FUNCTION_BLOCK "UNI_TO_GB2"   // FB9, SCL
{ S7_Optimized_Access := 'TRUE' }
VERSION : 0.1
   VAR_INPUT
      UNICODE : Word;
   END_VAR
   VAR_OUTPUT
      GB2312 : Word;
   END_VAR
   VAR
      UNI : Array[0..7480] of Word;
      GB2 : Array[0..7480] of Word;
   END_VAR
   VAR_TEMP
      i : UDInt;
      j : UDInt;
      li : UDInt;
      hi : UDInt;
   END_VAR
   // UNI[0] := 16#00A4;
   // UNI[1] := 16#00A7;
   // UNI[2] := 16#00A8;
   // UNI[3] := 16#00B0;
   // UNI[4] := 16#00B1;
   // UNI[5] := 16#00B7;
   // UNI[6] := 16#00D7;
   // UNI[7] := 16#00E0;
   // UNI[8] := 16#00E1;
   // UNI[9] := 16#00E8;
   // UNI[10] := 16#00E9;
   // UNI[11] := 16#00EA;
   // UNI[12] := 16#00EC;
   // UNI[13] := 16#00ED;
   // UNI[14] := 16#00F2;
   // UNI[15] := 16#00F3;
   // UNI[16] := 16#00F7;
   // UNI[17] := 16#00F9;
   // UNI[18] := 16#00FA;
   // UNI[19] := 16#00FC;
   // UNI[20] := 16#0101;
   // UNI[21] := 16#0113;
   // UNI[22] := 16#011B;
   // UNI[23] := 16#012B;
   // UNI[24] := 16#0144;
   // UNI[25] := 16#0148;
   // UNI[26] := 16#014D;
   // UNI[27] := 16#016B;
   // UNI[28] := 16#01CE;
   // UNI[29] := 16#01D0;
   // UNI[30] := 16#01D2;
   // UNI[31] := 16#01D4;
   // UNI[32] := 16#01D6;
   // UNI[33] := 16#01D8;
   // UNI[34] := 16#01DA;
   // UNI[35] := 16#01DC;
   // UNI[36] := 16#0251;
   // UNI[37] := 16#0261;
   // UNI[38] := 16#02C7;
   // UNI[39] := 16#02C9;
   // UNI[40] := 16#0391;
   // UNI[41] := 16#0392;
   // UNI[42] := 16#0393;
   // UNI[43] := 16#0394;
   // UNI[44] := 16#0395;
   // UNI[45] := 16#0396;
   // UNI[46] := 16#0397;
   // UNI[47] := 16#0398;
   // UNI[48] := 16#0399;
   // UNI[49] := 16#039A;
   // UNI[50] := 16#039B;
   // UNI[51] := 16#039C;
   // UNI[52] := 16#039D;
   // UNI[53] := 16#039E;
   // UNI[54] := 16#039F;
   // UNI[55] := 16#03A0;
   // UNI[56] := 16#03A1;
   // UNI[57] := 16#03A3;
   // UNI[58] := 16#03A4;
   // UNI[59] := 16#03A5;
   // UNI[60] := 16#03A6;
   // UNI[61] := 16#03A7;
   // UNI[62] := 16#03A8;
   // UNI[63] := 16#03A9;
   // UNI[64] := 16#03B1;
   // UNI[65] := 16#03B2;
   // UNI[66] := 16#03B3;
   // UNI[67] := 16#03B4;
   // UNI[68] := 16#03B5;
   // UNI[69] := 16#03B6;
   // UNI[70] := 16#03B7;
   // UNI[71] := 16#03B8;
   // UNI[72] := 16#03B9;
   // UNI[73] := 16#03BA;
   // UNI[74] := 16#03BB;
   // UNI[75] := 16#03BC;
   // UNI[76] := 16#03BD;
   // UNI[77] := 16#03BE;
   // UNI[78] := 16#03BF;
   // UNI[79] := 16#03C0;
   // UNI[80] := 16#03C1;
   // UNI[81] := 16#03C3;
   // UNI[82] := 16#03C4;
   // UNI[83] := 16#03C5;
   // UNI[84] := 16#03C6;
   // UNI[85] := 16#03C7;
   // UNI[86] := 16#03C8;
   // UNI[87] := 16#03C9;
   // UNI[88] := 16#0401;
   // UNI[89] := 16#0410;
   // UNI[90] := 16#0411;
   // UNI[91] := 16#0412;
   // UNI[92] := 16#0413;
   // UNI[93] := 16#0414;
   // UNI[94] := 16#0415;
   // UNI[95] := 16#0416;
   // UNI[96] := 16#0417;
   // UNI[97] := 16#0418;
   // UNI[98] := 16#0419;
   // UNI[99] := 16#041A;
   // UNI[100] := 16#041B;
   // UNI[101] := 16#041C;
   // UNI[102] := 16#041D;
   // UNI[103] := 16#041E;
   // UNI[104] := 16#041F;
   // UNI[105] := 16#0420;
   // UNI[106] := 16#0421;
   // UNI[107] := 16#0422;
   // UNI[108] := 16#0423;
   // UNI[109] := 16#0424;
   // UNI[110] := 16#0425;
   // UNI[111] := 16#0426;
   // UNI[112] := 16#0427;
   // UNI[113] := 16#0428;
   // UNI[114] := 16#0429;
   // UNI[115] := 16#042A;
   // UNI[116] := 16#042B;
   // UNI[117] := 16#042C;
   // UNI[118] := 16#042D;
   // UNI[119] := 16#042E;
   // UNI[120] := 16#042F;
   // UNI[121] := 16#0430;
   // UNI[122] := 16#0431;
   // UNI[123] := 16#0432;
   // UNI[124] := 16#0433;
   // UNI[125] := 16#0434;
   // UNI[126] := 16#0435;
   // UNI[127] := 16#0436;
   // UNI[128] := 16#0437;
   // UNI[129] := 16#0438;
   // UNI[130] := 16#0439;
   // UNI[131] := 16#043A;
   // UNI[132] := 16#043B;
   // UNI[133] := 16#043C;
   // UNI[134] := 16#043D;
   // UNI[135] := 16#043E;
   // UNI[136] := 16#043F;
   // UNI[137] := 16#0440;
   // UNI[138] := 16#0441;
   // UNI[139] := 16#0442;
   // UNI[140] := 16#0443;
   // UNI[141] := 16#0444;
   // UNI[142] := 16#0445;
   // UNI[143] := 16#0446;
   // UNI[144] := 16#0447;
   // UNI[145] := 16#0448;
   // UNI[146] := 16#0449;
   // UNI[147] := 16#044A;
   // UNI[148] := 16#044B;
   // UNI[149] := 16#044C;
   // UNI[150] := 16#044D;
   // UNI[151] := 16#044E;
   // UNI[152] := 16#044F;
   // UNI[153] := 16#0451;
   // UNI[154] := 16#2014;
   // UNI[155] := 16#2016;
   // UNI[156] := 16#2018;
   // UNI[157] := 16#2019;
   // UNI[158] := 16#201C;
   // UNI[159] := 16#201D;
   // UNI[160] := 16#2026;
   // UNI[161] := 16#2030;
   // UNI[162] := 16#2032;
   // UNI[163] := 16#2033;
   // UNI[164] := 16#203B;
   // UNI[165] := 16#2103;
   // UNI[166] := 16#2116;
   // UNI[167] := 16#2160;
   // UNI[168] := 16#2161;
   // UNI[169] := 16#2162;
   // UNI[170] := 16#2163;
   // UNI[171] := 16#2164;
   // UNI[172] := 16#2165;
   // UNI[173] := 16#2166;
   // UNI[174] := 16#2167;
   // UNI[175] := 16#2168;
   // UNI[176] := 16#2169;
   // UNI[177] := 16#216A;
   // UNI[178] := 16#216B;
   // UNI[179] := 16#2170;
   // UNI[180] := 16#2171;
   // UNI[181] := 16#2172;
   // UNI[182] := 16#2173;
   // UNI[183] := 16#2174;
   // UNI[184] := 16#2175;
   // UNI[185] := 16#2176;
   // UNI[186] := 16#2177;
   // UNI[187] := 16#2178;
   // UNI[188] := 16#2179;
   // UNI[189] := 16#2190;
   // UNI[190] := 16#2191;
   // UNI[191] := 16#2192;
   // UNI[192] := 16#2193;
   // UNI[193] := 16#2208;
   // UNI[194] := 16#220F;
   // UNI[195] := 16#2211;
   // UNI[196] := 16#221A;
   // UNI[197] := 16#221D;
   // UNI[198] := 16#221E;
   // UNI[199] := 16#2220;
   // UNI[200] := 16#2225;
   // UNI[201] := 16#2227;
   // UNI[202] := 16#2228;
   // UNI[203] := 16#2229;
   // UNI[204] := 16#222A;
   // UNI[205] := 16#222B;
   // UNI[206] := 16#222E;
   // UNI[207] := 16#2234;
   // UNI[208] := 16#2235;
   // UNI[209] := 16#2236;
   // UNI[210] := 16#2237;
   // UNI[211] := 16#223D;
   // UNI[212] := 16#2248;
   // UNI[213] := 16#224C;
   // UNI[214] := 16#2260;
   // UNI[215] := 16#2261;
   // UNI[216] := 16#2264;
   // UNI[217] := 16#2265;
   // UNI[218] := 16#226E;
   // UNI[219] := 16#226F;
   // UNI[220] := 16#2299;
   // UNI[221] := 16#22A5;
   // UNI[222] := 16#2312;
   // UNI[223] := 16#2460;
   // UNI[224] := 16#2461;
   // UNI[225] := 16#2462;
   // UNI[226] := 16#2463;
   // UNI[227] := 16#2464;
   // UNI[228] := 16#2465;
   // UNI[229] := 16#2466;
   // UNI[230] := 16#2467;
   // UNI[231] := 16#2468;
   // UNI[232] := 16#2469;
   // UNI[233] := 16#2474;
   // UNI[234] := 16#2475;
   // UNI[235] := 16#2476;
   // UNI[236] := 16#2477;
   // UNI[237] := 16#2478;
   // UNI[238] := 16#2479;
   // UNI[239] := 16#247A;
   // UNI[240] := 16#247B;
   // UNI[241] := 16#247C;
   // UNI[242] := 16#247D;
   // UNI[243] := 16#247E;
   // UNI[244] := 16#247F;
   // UNI[245] := 16#2480;
   // UNI[246] := 16#2481;
   // UNI[247] := 16#2482;
   // UNI[248] := 16#2483;
   // UNI[249] := 16#2484;
   // UNI[250] := 16#2485;
   // UNI[251] := 16#2486;
   // UNI[252] := 16#2487;
   // UNI[253] := 16#2488;
   // UNI[254] := 16#2489;
   // UNI[255] := 16#248A;
   // UNI[256] := 16#248B;
   // UNI[257] := 16#248C;
   // UNI[258] := 16#248D;
   // UNI[259] := 16#248E;
   // UNI[260] := 16#248F;
   // UNI[261] := 16#2490;
   // UNI[262] := 16#2491;
   // UNI[263] := 16#2492;
   // UNI[264] := 16#2493;
   // UNI[265] := 16#2494;
   // UNI[266] := 16#2495;
   // UNI[267] := 16#2496;
   // UNI[268] := 16#2497;
   // UNI[269] := 16#2498;
   // UNI[270] := 16#2499;
   // UNI[271] := 16#249A;
   // UNI[272] := 16#249B;
   // UNI[273] := 16#2500;
   // UNI[274] := 16#2501;
   // UNI[275] := 16#2502;
   // UNI[276] := 16#2503;
   // UNI[277] := 16#2504;
   // UNI[278] := 16#2505;
   // UNI[279] := 16#2506;
   // UNI[280] := 16#2507;
   // UNI[281] := 16#2508;
   // UNI[282] := 16#2509;
   // UNI[283] := 16#250A;
   // UNI[284] := 16#250B;
   // UNI[285] := 16#250C;
   // UNI[286] := 16#250D;
   // UNI[287] := 16#250E;
   // UNI[288] := 16#250F;
   // UNI[289] := 16#2510;
   // UNI[290] := 16#2511;
   // UNI[291] := 16#2512;
   // UNI[292] := 16#2513;
   // UNI[293] := 16#2514;
   // UNI[294] := 16#2515;
   // UNI[295] := 16#2516;
   // UNI[296] := 16#2517;
   // UNI[297] := 16#2518;
   // UNI[298] := 16#2519;
   // UNI[299] := 16#251A;
   // UNI[300] := 16#251B;
   // UNI[301] := 16#251C;
   // UNI[302] := 16#251D;
   // UNI[303] := 16#251E;
   // UNI[304] := 16#251F;
   // UNI[305] := 16#2520;
   // UNI[306] := 16#2521;
   // UNI[307] := 16#2522;
   // UNI[308] := 16#2523;
   // UNI[309] := 16#2524;
   // UNI[310] := 16#2525;
   // UNI[311] := 16#2526;
   // UNI[312] := 16#2527;
   // UNI[313] := 16#2528;
   // UNI[314] := 16#2529;
   // UNI[315] := 16#252A;
   // UNI[316] := 16#252B;
   // UNI[317] := 16#252C;
   // UNI[318] := 16#252D;
   // UNI[319] := 16#252E;
   // UNI[320] := 16#252F;
   // UNI[321] := 16#2530;
   // UNI[322] := 16#2531;
   // UNI[323] := 16#2532;
   // UNI[324] := 16#2533;
   // UNI[325] := 16#2534;
   // UNI[326] := 16#2535;
   // UNI[327] := 16#2536;
   // UNI[328] := 16#2537;
   // UNI[329] := 16#2538;
   // UNI[330] := 16#2539;
   // UNI[331] := 16#253A;
   // UNI[332] := 16#253B;
   // UNI[333] := 16#253C;
   // UNI[334] := 16#253D;
   // UNI[335] := 16#253E;
   // UNI[336] := 16#253F;
   // UNI[337] := 16#2540;
   // UNI[338] := 16#2541;
   // UNI[339] := 16#2542;
   // UNI[340] := 16#2543;
   // UNI[341] := 16#2544;
   // UNI[342] := 16#2545;
   // UNI[343] := 16#2546;
   // UNI[344] := 16#2547;
   // UNI[345] := 16#2548;
   // UNI[346] := 16#2549;
   // UNI[347] := 16#254A;
   // UNI[348] := 16#254B;
   // UNI[349] := 16#25A0;
   // UNI[350] := 16#25A1;
   // UNI[351] := 16#25B2;
   // UNI[352] := 16#25B3;
   // UNI[353] := 16#25C6;
   // UNI[354] := 16#25C7;
   // UNI[355] := 16#25CB;
   // UNI[356] := 16#25CE;
   // UNI[357] := 16#25CF;
   // UNI[358] := 16#2605;
   // UNI[359] := 16#2606;
   // UNI[360] := 16#2640;
   // UNI[361] := 16#2642;
   // UNI[362] := 16#3000;
   // UNI[363] := 16#3001;
   // UNI[364] := 16#3002;
   // UNI[365] := 16#3003;
   // UNI[366] := 16#3005;
   // UNI[367] := 16#3008;
   // UNI[368] := 16#3009;
   // UNI[369] := 16#300A;
   // UNI[370] := 16#300B;
   // UNI[371] := 16#300C;
   // UNI[372] := 16#300D;
   // UNI[373] := 16#300E;
   // UNI[374] := 16#300F;
   // UNI[375] := 16#3010;
   // UNI[376] := 16#3011;
   // UNI[377] := 16#3013;
   // UNI[378] := 16#3014;
   // UNI[379] := 16#3015;
   // UNI[380] := 16#3016;
   // UNI[381] := 16#3017;
   // UNI[382] := 16#3041;
   // UNI[383] := 16#3042;
   // UNI[384] := 16#3043;
   // UNI[385] := 16#3044;
   // UNI[386] := 16#3045;
   // UNI[387] := 16#3046;
   // UNI[388] := 16#3047;
   // UNI[389] := 16#3048;
   // UNI[390] := 16#3049;
   // UNI[391] := 16#304A;
   // UNI[392] := 16#304B;
   // UNI[393] := 16#304C;
   // UNI[394] := 16#304D;
   // UNI[395] := 16#304E;
   // UNI[396] := 16#304F;
   // UNI[397] := 16#3050;
   // UNI[398] := 16#3051;
   // UNI[399] := 16#3052;
   // UNI[400] := 16#3053;
   // UNI[401] := 16#3054;
   // UNI[402] := 16#3055;
   // UNI[403] := 16#3056;
   // UNI[404] := 16#3057;
   // UNI[405] := 16#3058;
   // UNI[406] := 16#3059;
   // UNI[407] := 16#305A;
   // UNI[408] := 16#305B;
   // UNI[409] := 16#305C;
   // UNI[410] := 16#305D;
   // UNI[411] := 16#305E;
   // UNI[412] := 16#305F;
   // UNI[413] := 16#3060;
   // UNI[414] := 16#3061;
   // UNI[415] := 16#3062;
   // UNI[416] := 16#3063;
   // UNI[417] := 16#3064;
   // UNI[418] := 16#3065;
   // UNI[419] := 16#3066;
   // UNI[420] := 16#3067;
   // UNI[421] := 16#3068;
   // UNI[422] := 16#3069;
   // UNI[423] := 16#306A;
   // UNI[424] := 16#306B;
   // UNI[425] := 16#306C;
   // UNI[426] := 16#306D;
   // UNI[427] := 16#306E;
   // UNI[428] := 16#306F;
   // UNI[429] := 16#3070;
   // UNI[430] := 16#3071;
   // UNI[431] := 16#3072;
   // UNI[432] := 16#3073;
   // UNI[433] := 16#3074;
   // UNI[434] := 16#3075;
   // UNI[435] := 16#3076;
   // UNI[436] := 16#3077;
   // UNI[437] := 16#3078;
   // UNI[438] := 16#3079;
   // UNI[439] := 16#307A;
   // UNI[440] := 16#307B;
   // UNI[441] := 16#307C;
   // UNI[442] := 16#307D;
   // UNI[443] := 16#307E;
   // UNI[444] := 16#307F;
   // UNI[445] := 16#3080;
   // UNI[446] := 16#3081;
   // UNI[447] := 16#3082;
   // UNI[448] := 16#3083;
   // UNI[449] := 16#3084;
   // UNI[450] := 16#3085;
   // UNI[451] := 16#3086;
   // UNI[452] := 16#3087;
   // UNI[453] := 16#3088;
   // UNI[454] := 16#3089;
   // UNI[455] := 16#308A;
   // UNI[456] := 16#308B;
   // UNI[457] := 16#308C;
   // UNI[458] := 16#308D;
   // UNI[459] := 16#308E;
   // UNI[460] := 16#308F;
   // UNI[461] := 16#3090;
   // UNI[462] := 16#3091;
   // UNI[463] := 16#3092;
   // UNI[464] := 16#3093;
   // UNI[465] := 16#30A1;
   // UNI[466] := 16#30A2;
   // UNI[467] := 16#30A3;
   // UNI[468] := 16#30A4;
   // UNI[469] := 16#30A5;
   // UNI[470] := 16#30A6;
   // UNI[471] := 16#30A7;
   // UNI[472] := 16#30A8;
   // UNI[473] := 16#30A9;
   // UNI[474] := 16#30AA;
   // UNI[475] := 16#30AB;
   // UNI[476] := 16#30AC;
   // UNI[477] := 16#30AD;
   // UNI[478] := 16#30AE;
   // UNI[479] := 16#30AF;
   // UNI[480] := 16#30B0;
   // UNI[481] := 16#30B1;
   // UNI[482] := 16#30B2;
   // UNI[483] := 16#30B3;
   // UNI[484] := 16#30B4;
   // UNI[485] := 16#30B5;
   // UNI[486] := 16#30B6;
   // UNI[487] := 16#30B7;
   // UNI[488] := 16#30B8;
   // UNI[489] := 16#30B9;
   // UNI[490] := 16#30BA;
   // UNI[491] := 16#30BB;
   // UNI[492] := 16#30BC;
   // UNI[493] := 16#30BD;
   // UNI[494] := 16#30BE;
   // UNI[495] := 16#30BF;
   // UNI[496] := 16#30C0;
   // UNI[497] := 16#30C1;
   // UNI[498] := 16#30C2;
   // UNI[499] := 16#30C3;
   // UNI[500] := 16#30C4;
   // UNI[501] := 16#30C5;
   // UNI[502] := 16#30C6;
   // UNI[503] := 16#30C7;
   // UNI[504] := 16#30C8;
   // UNI[505] := 16#30C9;
   // UNI[506] := 16#30CA;
   // UNI[507] := 16#30CB;
   // UNI[508] := 16#30CC;
   // UNI[509] := 16#30CD;
   // UNI[510] := 16#30CE;
   // UNI[511] := 16#30CF;
   // UNI[512] := 16#30D0;
   // UNI[513] := 16#30D1;
   // UNI[514] := 16#30D2;
   // UNI[515] := 16#30D3;
   // UNI[516] := 16#30D4;
   // UNI[517] := 16#30D5;
   // UNI[518] := 16#30D6;
   // UNI[519] := 16#30D7;
   // UNI[520] := 16#30D8;
   // UNI[521] := 16#30D9;
   // UNI[522] := 16#30DA;
   // UNI[523] := 16#30DB;
   // UNI[524] := 16#30DC;
   // UNI[525] := 16#30DD;
   // UNI[526] := 16#30DE;
   // UNI[527] := 16#30DF;
   // UNI[528] := 16#30E0;
   // UNI[529] := 16#30E1;
   // UNI[530] := 16#30E2;
   // UNI[531] := 16#30E3;
   // UNI[532] := 16#30E4;
   // UNI[533] := 16#30E5;
   // UNI[534] := 16#30E6;
   // UNI[535] := 16#30E7;
   // UNI[536] := 16#30E8;
   // UNI[537] := 16#30E9;
   // UNI[538] := 16#30EA;
   // UNI[539] := 16#30EB;
   // UNI[540] := 16#30EC;
   // UNI[541] := 16#30ED;
   // UNI[542] := 16#30EE;
   // UNI[543] := 16#30EF;
   // UNI[544] := 16#30F0;
   // UNI[545] := 16#30F1;
   // UNI[546] := 16#30F2;
   // UNI[547] := 16#30F3;
   // UNI[548] := 16#30F4;
   // UNI[549] := 16#30F5;
   // UNI[550] := 16#30F6;
   // UNI[551] := 16#3105;
   // UNI[552] := 16#3106;
   // UNI[553] := 16#3107;
   // UNI[554] := 16#3108;
   // UNI[555] := 16#3109;
   // UNI[556] := 16#310A;
   // UNI[557] := 16#310B;
   // UNI[558] := 16#310C;
   // UNI[559] := 16#310D;
   // UNI[560] := 16#310E;
   // UNI[561] := 16#310F;
   // UNI[562] := 16#3110;
   // UNI[563] := 16#3111;
   // UNI[564] := 16#3112;
   // UNI[565] := 16#3113;
   // UNI[566] := 16#3114;
   // UNI[567] := 16#3115;
   // UNI[568] := 16#3116;
   // UNI[569] := 16#3117;
   // UNI[570] := 16#3118;
   // UNI[571] := 16#3119;
   // UNI[572] := 16#311A;
   // UNI[573] := 16#311B;
   // UNI[574] := 16#311C;
   // UNI[575] := 16#311D;
   // UNI[576] := 16#311E;
   // UNI[577] := 16#311F;
   // UNI[578] := 16#3120;
   // UNI[579] := 16#3121;
   // UNI[580] := 16#3122;
   // UNI[581] := 16#3123;
   // UNI[582] := 16#3124;
   // UNI[583] := 16#3125;
   // UNI[584] := 16#3126;
   // UNI[585] := 16#3127;
   // UNI[586] := 16#3128;
   // UNI[587] := 16#3129;
   // UNI[588] := 16#3220;
   // UNI[589] := 16#3221;
   // UNI[590] := 16#3222;
   // UNI[591] := 16#3223;
   // UNI[592] := 16#3224;
   // UNI[593] := 16#3225;
   // UNI[594] := 16#3226;
   // UNI[595] := 16#3227;
   // UNI[596] := 16#3228;
   // UNI[597] := 16#3229;
   // UNI[598] := 16#4E00;
   // UNI[599] := 16#4E01;
   // UNI[600] := 16#4E03;
   // UNI[601] := 16#4E07;
   // UNI[602] := 16#4E08;
   // UNI[603] := 16#4E09;
   // UNI[604] := 16#4E0A;
   // UNI[605] := 16#4E0B;
   // UNI[606] := 16#4E0C;
   // UNI[607] := 16#4E0D;
   // UNI[608] := 16#4E0E;
   // UNI[609] := 16#4E10;
   // UNI[610] := 16#4E11;
   // UNI[611] := 16#4E13;
   // UNI[612] := 16#4E14;
   // UNI[613] := 16#4E15;
   // UNI[614] := 16#4E16;
   // UNI[615] := 16#4E18;
   // UNI[616] := 16#4E19;
   // UNI[617] := 16#4E1A;
   // UNI[618] := 16#4E1B;
   // UNI[619] := 16#4E1C;
   // UNI[620] := 16#4E1D;
   // UNI[621] := 16#4E1E;
   // UNI[622] := 16#4E22;
   // UNI[623] := 16#4E24;
   // UNI[624] := 16#4E25;
   // UNI[625] := 16#4E27;
   // UNI[626] := 16#4E28;
   // UNI[627] := 16#4E2A;
   // UNI[628] := 16#4E2B;
   // UNI[629] := 16#4E2C;
   // UNI[630] := 16#4E2D;
   // UNI[631] := 16#4E30;
   // UNI[632] := 16#4E32;
   // UNI[633] := 16#4E34;
   // UNI[634] := 16#4E36;
   // UNI[635] := 16#4E38;
   // UNI[636] := 16#4E39;
   // UNI[637] := 16#4E3A;
   // UNI[638] := 16#4E3B;
   // UNI[639] := 16#4E3D;
   // UNI[640] := 16#4E3E;
   // UNI[641] := 16#4E3F;
   // UNI[642] := 16#4E43;
   // UNI[643] := 16#4E45;
   // UNI[644] := 16#4E47;
   // UNI[645] := 16#4E48;
   // UNI[646] := 16#4E49;
   // UNI[647] := 16#4E4B;
   // UNI[648] := 16#4E4C;
   // UNI[649] := 16#4E4D;
   // UNI[650] := 16#4E4E;
   // UNI[651] := 16#4E4F;
   // UNI[652] := 16#4E50;
   // UNI[653] := 16#4E52;
   // UNI[654] := 16#4E53;
   // UNI[655] := 16#4E54;
   // UNI[656] := 16#4E56;
   // UNI[657] := 16#4E58;
   // UNI[658] := 16#4E59;
   // UNI[659] := 16#4E5C;
   // UNI[660] := 16#4E5D;
   // UNI[661] := 16#4E5E;
   // UNI[662] := 16#4E5F;
   // UNI[663] := 16#4E60;
   // UNI[664] := 16#4E61;
   // UNI[665] := 16#4E66;
   // UNI[666] := 16#4E69;
   // UNI[667] := 16#4E70;
   // UNI[668] := 16#4E71;
   // UNI[669] := 16#4E73;
   // UNI[670] := 16#4E7E;
   // UNI[671] := 16#4E86;
   // UNI[672] := 16#4E88;
   // UNI[673] := 16#4E89;
   // UNI[674] := 16#4E8B;
   // UNI[675] := 16#4E8C;
   // UNI[676] := 16#4E8D;
   // UNI[677] := 16#4E8E;
   // UNI[678] := 16#4E8F;
   // UNI[679] := 16#4E91;
   // UNI[680] := 16#4E92;
   // UNI[681] := 16#4E93;
   // UNI[682] := 16#4E94;
   // UNI[683] := 16#4E95;
   // UNI[684] := 16#4E98;
   // UNI[685] := 16#4E9A;
   // UNI[686] := 16#4E9B;
   // UNI[687] := 16#4E9F;
   // UNI[688] := 16#4EA0;
   // UNI[689] := 16#4EA1;
   // UNI[690] := 16#4EA2;
   // UNI[691] := 16#4EA4;
   // UNI[692] := 16#4EA5;
   // UNI[693] := 16#4EA6;
   // UNI[694] := 16#4EA7;
   // UNI[695] := 16#4EA8;
   // UNI[696] := 16#4EA9;
   // UNI[697] := 16#4EAB;
   // UNI[698] := 16#4EAC;
   // UNI[699] := 16#4EAD;
   // UNI[700] := 16#4EAE;
   // UNI[701] := 16#4EB2;
   // UNI[702] := 16#4EB3;
   // UNI[703] := 16#4EB5;
   // UNI[704] := 16#4EBA;
   // UNI[705] := 16#4EBB;
   // UNI[706] := 16#4EBF;
   // UNI[707] := 16#4EC0;
   // UNI[708] := 16#4EC1;
   // UNI[709] := 16#4EC2;
   // UNI[710] := 16#4EC3;
   // UNI[711] := 16#4EC4;
   // UNI[712] := 16#4EC5;
   // UNI[713] := 16#4EC6;
   // UNI[714] := 16#4EC7;
   // UNI[715] := 16#4EC9;
   // UNI[716] := 16#4ECA;
   // UNI[717] := 16#4ECB;
   // UNI[718] := 16#4ECD;
   // UNI[719] := 16#4ECE;
   // UNI[720] := 16#4ED1;
   // UNI[721] := 16#4ED3;
   // UNI[722] := 16#4ED4;
   // UNI[723] := 16#4ED5;
   // UNI[724] := 16#4ED6;
   // UNI[725] := 16#4ED7;
   // UNI[726] := 16#4ED8;
   // UNI[727] := 16#4ED9;
   // UNI[728] := 16#4EDD;
   // UNI[729] := 16#4EDE;
   // UNI[730] := 16#4EDF;
   // UNI[731] := 16#4EE1;
   // UNI[732] := 16#4EE3;
   // UNI[733] := 16#4EE4;
   // UNI[734] := 16#4EE5;
   // UNI[735] := 16#4EE8;
   // UNI[736] := 16#4EEA;
   // UNI[737] := 16#4EEB;
   // UNI[738] := 16#4EEC;
   // UNI[739] := 16#4EF0;
   // UNI[740] := 16#4EF2;
   // UNI[741] := 16#4EF3;
   // UNI[742] := 16#4EF5;
   // UNI[743] := 16#4EF6;
   // UNI[744] := 16#4EF7;
   // UNI[745] := 16#4EFB;
   // UNI[746] := 16#4EFD;
   // UNI[747] := 16#4EFF;
   // UNI[748] := 16#4F01;
   // UNI[749] := 16#4F09;
   // UNI[750] := 16#4F0A;
   // UNI[751] := 16#4F0D;
   // UNI[752] := 16#4F0E;
   // UNI[753] := 16#4F0F;
   // UNI[754] := 16#4F10;
   // UNI[755] := 16#4F11;
   // UNI[756] := 16#4F17;
   // UNI[757] := 16#4F18;
   // UNI[758] := 16#4F19;
   // UNI[759] := 16#4F1A;
   // UNI[760] := 16#4F1B;
   // UNI[761] := 16#4F1E;
   // UNI[762] := 16#4F1F;
   // UNI[763] := 16#4F20;
   // UNI[764] := 16#4F22;
   // UNI[765] := 16#4F24;
   // UNI[766] := 16#4F25;
   // UNI[767] := 16#4F26;
   // UNI[768] := 16#4F27;
   // UNI[769] := 16#4F2A;
   // UNI[770] := 16#4F2B;
   // UNI[771] := 16#4F2F;
   // UNI[772] := 16#4F30;
   // UNI[773] := 16#4F32;
   // UNI[774] := 16#4F34;
   // UNI[775] := 16#4F36;
   // UNI[776] := 16#4F38;
   // UNI[777] := 16#4F3A;
   // UNI[778] := 16#4F3C;
   // UNI[779] := 16#4F3D;
   // UNI[780] := 16#4F43;
   // UNI[781] := 16#4F46;
   // UNI[782] := 16#4F4D;
   // UNI[783] := 16#4F4E;
   // UNI[784] := 16#4F4F;
   // UNI[785] := 16#4F50;
   // UNI[786] := 16#4F51;
   // UNI[787] := 16#4F53;
   // UNI[788] := 16#4F55;
   // UNI[789] := 16#4F57;
   // UNI[790] := 16#4F58;
   // UNI[791] := 16#4F59;
   // UNI[792] := 16#4F5A;
   // UNI[793] := 16#4F5B;
   // UNI[794] := 16#4F5C;
   // UNI[795] := 16#4F5D;
   // UNI[796] := 16#4F5E;
   // UNI[797] := 16#4F5F;
   // UNI[798] := 16#4F60;
   // UNI[799] := 16#4F63;
   // UNI[800] := 16#4F64;
   // UNI[801] := 16#4F65;
   // UNI[802] := 16#4F67;
   // UNI[803] := 16#4F69;
   // UNI[804] := 16#4F6C;
   // UNI[805] := 16#4F6F;
   // UNI[806] := 16#4F70;
   // UNI[807] := 16#4F73;
   // UNI[808] := 16#4F74;
   // UNI[809] := 16#4F76;
   // UNI[810] := 16#4F7B;
   // UNI[811] := 16#4F7C;
   // UNI[812] := 16#4F7E;
   // UNI[813] := 16#4F7F;
   // UNI[814] := 16#4F83;
   // UNI[815] := 16#4F84;
   // UNI[816] := 16#4F88;
   // UNI[817] := 16#4F89;
   // UNI[818] := 16#4F8B;
   // UNI[819] := 16#4F8D;
   // UNI[820] := 16#4F8F;
   // UNI[821] := 16#4F91;
   // UNI[822] := 16#4F94;
   // UNI[823] := 16#4F97;
   // UNI[824] := 16#4F9B;
   // UNI[825] := 16#4F9D;
   // UNI[826] := 16#4FA0;
   // UNI[827] := 16#4FA3;
   // UNI[828] := 16#4FA5;
   // UNI[829] := 16#4FA6;
   // UNI[830] := 16#4FA7;
   // UNI[831] := 16#4FA8;
   // UNI[832] := 16#4FA9;
   // UNI[833] := 16#4FAA;
   // UNI[834] := 16#4FAC;
   // UNI[835] := 16#4FAE;
   // UNI[836] := 16#4FAF;
   // UNI[837] := 16#4FB5;
   // UNI[838] := 16#4FBF;
   // UNI[839] := 16#4FC3;
   // UNI[840] := 16#4FC4;
   // UNI[841] := 16#4FC5;
   // UNI[842] := 16#4FCA;
   // UNI[843] := 16#4FCE;
   // UNI[844] := 16#4FCF;
   // UNI[845] := 16#4FD0;
   // UNI[846] := 16#4FD1;
   // UNI[847] := 16#4FD7;
   // UNI[848] := 16#4FD8;
   // UNI[849] := 16#4FDA;
   // UNI[850] := 16#4FDC;
   // UNI[851] := 16#4FDD;
   // UNI[852] := 16#4FDE;
   // UNI[853] := 16#4FDF;
   // UNI[854] := 16#4FE1;
   // UNI[855] := 16#4FE3;
   // UNI[856] := 16#4FE6;
   // UNI[857] := 16#4FE8;
   // UNI[858] := 16#4FE9;
   // UNI[859] := 16#4FEA;
   // UNI[860] := 16#4FED;
   // UNI[861] := 16#4FEE;
   // UNI[862] := 16#4FEF;
   // UNI[863] := 16#4FF1;
   // UNI[864] := 16#4FF3;
   // UNI[865] := 16#4FF8;
   // UNI[866] := 16#4FFA;
   // UNI[867] := 16#4FFE;
   // UNI[868] := 16#500C;
   // UNI[869] := 16#500D;
   // UNI[870] := 16#500F;
   // UNI[871] := 16#5012;
   // UNI[872] := 16#5014;
   // UNI[873] := 16#5018;
   // UNI[874] := 16#5019;
   // UNI[875] := 16#501A;
   // UNI[876] := 16#501C;
   // UNI[877] := 16#501F;
   // UNI[878] := 16#5021;
   // UNI[879] := 16#5025;
   // UNI[880] := 16#5026;
   // UNI[881] := 16#5028;
   // UNI[882] := 16#5029;
   // UNI[883] := 16#502A;
   // UNI[884] := 16#502C;
   // UNI[885] := 16#502D;
   // UNI[886] := 16#502E;
   // UNI[887] := 16#503A;
   // UNI[888] := 16#503C;
   // UNI[889] := 16#503E;
   // UNI[890] := 16#5043;
   // UNI[891] := 16#5047;
   // UNI[892] := 16#5048;
   // UNI[893] := 16#504C;
   // UNI[894] := 16#504E;
   // UNI[895] := 16#504F;
   // UNI[896] := 16#5055;
   // UNI[897] := 16#505A;
   // UNI[898] := 16#505C;
   // UNI[899] := 16#5065;
   // UNI[900] := 16#506C;
   // UNI[901] := 16#5076;
   // UNI[902] := 16#5077;
   // UNI[903] := 16#507B;
   // UNI[904] := 16#507E;
   // UNI[905] := 16#507F;
   // UNI[906] := 16#5080;
   // UNI[907] := 16#5085;
   // UNI[908] := 16#5088;
   // UNI[909] := 16#508D;
   // UNI[910] := 16#50A3;
   // UNI[911] := 16#50A5;
   // UNI[912] := 16#50A7;
   // UNI[913] := 16#50A8;
   // UNI[914] := 16#50A9;
   // UNI[915] := 16#50AC;
   // UNI[916] := 16#50B2;
   // UNI[917] := 16#50BA;
   // UNI[918] := 16#50BB;
   // UNI[919] := 16#50CF;
   // UNI[920] := 16#50D6;
   // UNI[921] := 16#50DA;
   // UNI[922] := 16#50E6;
   // UNI[923] := 16#50E7;
   // UNI[924] := 16#50EC;
   // UNI[925] := 16#50ED;
   // UNI[926] := 16#50EE;
   // UNI[927] := 16#50F3;
   // UNI[928] := 16#50F5;
   // UNI[929] := 16#50FB;
   // UNI[930] := 16#5106;
   // UNI[931] := 16#5107;
   // UNI[932] := 16#510B;
   // UNI[933] := 16#5112;
   // UNI[934] := 16#5121;
   // UNI[935] := 16#513F;
   // UNI[936] := 16#5140;
   // UNI[937] := 16#5141;
   // UNI[938] := 16#5143;
   // UNI[939] := 16#5144;
   // UNI[940] := 16#5145;
   // UNI[941] := 16#5146;
   // UNI[942] := 16#5148;
   // UNI[943] := 16#5149;
   // UNI[944] := 16#514B;
   // UNI[945] := 16#514D;
   // UNI[946] := 16#5151;
   // UNI[947] := 16#5154;
   // UNI[948] := 16#5155;
   // UNI[949] := 16#5156;
   // UNI[950] := 16#515A;
   // UNI[951] := 16#515C;
   // UNI[952] := 16#5162;
   // UNI[953] := 16#5165;
   // UNI[954] := 16#5168;
   // UNI[955] := 16#516B;
   // UNI[956] := 16#516C;
   // UNI[957] := 16#516D;
   // UNI[958] := 16#516E;
   // UNI[959] := 16#5170;
   // UNI[960] := 16#5171;
   // UNI[961] := 16#5173;
   // UNI[962] := 16#5174;
   // UNI[963] := 16#5175;
   // UNI[964] := 16#5176;
   // UNI[965] := 16#5177;
   // UNI[966] := 16#5178;
   // UNI[967] := 16#5179;
   // UNI[968] := 16#517B;
   // UNI[969] := 16#517C;
   // UNI[970] := 16#517D;
   // UNI[971] := 16#5180;
   // UNI[972] := 16#5181;
   // UNI[973] := 16#5182;
   // UNI[974] := 16#5185;
   // UNI[975] := 16#5188;
   // UNI[976] := 16#5189;
   // UNI[977] := 16#518C;
   // UNI[978] := 16#518D;
   // UNI[979] := 16#5192;
   // UNI[980] := 16#5195;
   // UNI[981] := 16#5196;
   // UNI[982] := 16#5197;
   // UNI[983] := 16#5199;
   // UNI[984] := 16#519B;
   // UNI[985] := 16#519C;
   // UNI[986] := 16#51A0;
   // UNI[987] := 16#51A2;
   // UNI[988] := 16#51A4;
   // UNI[989] := 16#51A5;
   // UNI[990] := 16#51AB;
   // UNI[991] := 16#51AC;
   // UNI[992] := 16#51AF;
   // UNI[993] := 16#51B0;
   // UNI[994] := 16#51B1;
   // UNI[995] := 16#51B2;
   // UNI[996] := 16#51B3;
   // UNI[997] := 16#51B5;
   // UNI[998] := 16#51B6;
   // UNI[999] := 16#51B7;
   // UNI[1000] := 16#51BB;
   // UNI[1001] := 16#51BC;
   // UNI[1002] := 16#51BD;
   // UNI[1003] := 16#51C0;
   // UNI[1004] := 16#51C4;
   // UNI[1005] := 16#51C6;
   // UNI[1006] := 16#51C7;
   // UNI[1007] := 16#51C9;
   // UNI[1008] := 16#51CB;
   // UNI[1009] := 16#51CC;
   // UNI[1010] := 16#51CF;
   // UNI[1011] := 16#51D1;
   // UNI[1012] := 16#51DB;
   // UNI[1013] := 16#51DD;
   // UNI[1014] := 16#51E0;
   // UNI[1015] := 16#51E1;
   // UNI[1016] := 16#51E4;
   // UNI[1017] := 16#51EB;
   // UNI[1018] := 16#51ED;
   // UNI[1019] := 16#51EF;
   // UNI[1020] := 16#51F0;
   // UNI[1021] := 16#51F3;
   // UNI[1022] := 16#51F5;
   // UNI[1023] := 16#51F6;
   // UNI[1024] := 16#51F8;
   // UNI[1025] := 16#51F9;
   // UNI[1026] := 16#51FA;
   // UNI[1027] := 16#51FB;
   // UNI[1028] := 16#51FC;
   // UNI[1029] := 16#51FD;
   // UNI[1030] := 16#51FF;
   // UNI[1031] := 16#5200;
   // UNI[1032] := 16#5201;
   // UNI[1033] := 16#5202;
   // UNI[1034] := 16#5203;
   // UNI[1035] := 16#5206;
   // UNI[1036] := 16#5207;
   // UNI[1037] := 16#5208;
   // UNI[1038] := 16#520A;
   // UNI[1039] := 16#520D;
   // UNI[1040] := 16#520E;
   // UNI[1041] := 16#5211;
   // UNI[1042] := 16#5212;
   // UNI[1043] := 16#5216;
   // UNI[1044] := 16#5217;
   // UNI[1045] := 16#5218;
   // UNI[1046] := 16#5219;
   // UNI[1047] := 16#521A;
   // UNI[1048] := 16#521B;
   // UNI[1049] := 16#521D;
   // UNI[1050] := 16#5220;
   // UNI[1051] := 16#5224;
   // UNI[1052] := 16#5228;
   // UNI[1053] := 16#5229;
   // UNI[1054] := 16#522B;
   // UNI[1055] := 16#522D;
   // UNI[1056] := 16#522E;
   // UNI[1057] := 16#5230;
   // UNI[1058] := 16#5233;
   // UNI[1059] := 16#5236;
   // UNI[1060] := 16#5237;
   // UNI[1061] := 16#5238;
   // UNI[1062] := 16#5239;
   // UNI[1063] := 16#523A;
   // UNI[1064] := 16#523B;
   // UNI[1065] := 16#523D;
   // UNI[1066] := 16#523F;
   // UNI[1067] := 16#5240;
   // UNI[1068] := 16#5241;
   // UNI[1069] := 16#5242;
   // UNI[1070] := 16#5243;
   // UNI[1071] := 16#524A;
   // UNI[1072] := 16#524C;
   // UNI[1073] := 16#524D;
   // UNI[1074] := 16#5250;
   // UNI[1075] := 16#5251;
   // UNI[1076] := 16#5254;
   // UNI[1077] := 16#5256;
   // UNI[1078] := 16#525C;
   // UNI[1079] := 16#525E;
   // UNI[1080] := 16#5261;
   // UNI[1081] := 16#5265;
   // UNI[1082] := 16#5267;
   // UNI[1083] := 16#5269;
   // UNI[1084] := 16#526A;
   // UNI[1085] := 16#526F;
   // UNI[1086] := 16#5272;
   // UNI[1087] := 16#527D;
   // UNI[1088] := 16#527F;
   // UNI[1089] := 16#5281;
   // UNI[1090] := 16#5282;
   // UNI[1091] := 16#5288;
   // UNI[1092] := 16#5290;
   // UNI[1093] := 16#5293;
   // UNI[1094] := 16#529B;
   // UNI[1095] := 16#529D;
   // UNI[1096] := 16#529E;
   // UNI[1097] := 16#529F;
   // UNI[1098] := 16#52A0;
   // UNI[1099] := 16#52A1;
   // UNI[1100] := 16#52A2;
   // UNI[1101] := 16#52A3;
   // UNI[1102] := 16#52A8;
   // UNI[1103] := 16#52A9;
   // UNI[1104] := 16#52AA;
   // UNI[1105] := 16#52AB;
   // UNI[1106] := 16#52AC;
   // UNI[1107] := 16#52AD;
   // UNI[1108] := 16#52B1;
   // UNI[1109] := 16#52B2;
   // UNI[1110] := 16#52B3;
   // UNI[1111] := 16#52BE;
   // UNI[1112] := 16#52BF;
   // UNI[1113] := 16#52C3;
   // UNI[1114] := 16#52C7;
   // UNI[1115] := 16#52C9;
   // UNI[1116] := 16#52CB;
   // UNI[1117] := 16#52D0;
   // UNI[1118] := 16#52D2;
   // UNI[1119] := 16#52D6;
   // UNI[1120] := 16#52D8;
   // UNI[1121] := 16#52DF;
   // UNI[1122] := 16#52E4;
   // UNI[1123] := 16#52F0;
   // UNI[1124] := 16#52F9;
   // UNI[1125] := 16#52FA;
   // UNI[1126] := 16#52FE;
   // UNI[1127] := 16#52FF;
   // UNI[1128] := 16#5300;
   // UNI[1129] := 16#5305;
   // UNI[1130] := 16#5306;
   // UNI[1131] := 16#5308;
   // UNI[1132] := 16#530D;
   // UNI[1133] := 16#530F;
   // UNI[1134] := 16#5310;
   // UNI[1135] := 16#5315;
   // UNI[1136] := 16#5316;
   // UNI[1137] := 16#5317;
   // UNI[1138] := 16#5319;
   // UNI[1139] := 16#531A;
   // UNI[1140] := 16#531D;
   // UNI[1141] := 16#5320;
   // UNI[1142] := 16#5321;
   // UNI[1143] := 16#5323;
   // UNI[1144] := 16#5326;
   // UNI[1145] := 16#532A;
   // UNI[1146] := 16#532E;
   // UNI[1147] := 16#5339;
   // UNI[1148] := 16#533A;
   // UNI[1149] := 16#533B;
   // UNI[1150] := 16#533E;
   // UNI[1151] := 16#533F;
   // UNI[1152] := 16#5341;
   // UNI[1153] := 16#5343;
   // UNI[1154] := 16#5345;
   // UNI[1155] := 16#5347;
   // UNI[1156] := 16#5348;
   // UNI[1157] := 16#5349;
   // UNI[1158] := 16#534A;
   // UNI[1159] := 16#534E;
   // UNI[1160] := 16#534F;
   // UNI[1161] := 16#5351;
   // UNI[1162] := 16#5352;
   // UNI[1163] := 16#5353;
   // UNI[1164] := 16#5355;
   // UNI[1165] := 16#5356;
   // UNI[1166] := 16#5357;
   // UNI[1167] := 16#535A;
   // UNI[1168] := 16#535C;
   // UNI[1169] := 16#535E;
   // UNI[1170] := 16#535F;
   // UNI[1171] := 16#5360;
   // UNI[1172] := 16#5361;
   // UNI[1173] := 16#5362;
   // UNI[1174] := 16#5363;
   // UNI[1175] := 16#5364;
   // UNI[1176] := 16#5366;
   // UNI[1177] := 16#5367;
   // UNI[1178] := 16#5369;
   // UNI[1179] := 16#536B;
   // UNI[1180] := 16#536E;
   // UNI[1181] := 16#536F;
   // UNI[1182] := 16#5370;
   // UNI[1183] := 16#5371;
   // UNI[1184] := 16#5373;
   // UNI[1185] := 16#5374;
   // UNI[1186] := 16#5375;
   // UNI[1187] := 16#5377;
   // UNI[1188] := 16#5378;
   // UNI[1189] := 16#537A;
   // UNI[1190] := 16#537F;
   // UNI[1191] := 16#5382;
   // UNI[1192] := 16#5384;
   // UNI[1193] := 16#5385;
   // UNI[1194] := 16#5386;
   // UNI[1195] := 16#5389;
   // UNI[1196] := 16#538B;
   // UNI[1197] := 16#538C;
   // UNI[1198] := 16#538D;
   // UNI[1199] := 16#5395;
   // UNI[1200] := 16#5398;
   // UNI[1201] := 16#539A;
   // UNI[1202] := 16#539D;
   // UNI[1203] := 16#539F;
   // UNI[1204] := 16#53A2;
   // UNI[1205] := 16#53A3;
   // UNI[1206] := 16#53A5;
   // UNI[1207] := 16#53A6;
   // UNI[1208] := 16#53A8;
   // UNI[1209] := 16#53A9;
   // UNI[1210] := 16#53AE;
   // UNI[1211] := 16#53B6;
   // UNI[1212] := 16#53BB;
   // UNI[1213] := 16#53BF;
   // UNI[1214] := 16#53C1;
   // UNI[1215] := 16#53C2;
   // UNI[1216] := 16#53C8;
   // UNI[1217] := 16#53C9;
   // UNI[1218] := 16#53CA;
   // UNI[1219] := 16#53CB;
   // UNI[1220] := 16#53CC;
   // UNI[1221] := 16#53CD;
   // UNI[1222] := 16#53D1;
   // UNI[1223] := 16#53D4;
   // UNI[1224] := 16#53D6;
   // UNI[1225] := 16#53D7;
   // UNI[1226] := 16#53D8;
   // UNI[1227] := 16#53D9;
   // UNI[1228] := 16#53DB;
   // UNI[1229] := 16#53DF;
   // UNI[1230] := 16#53E0;
   // UNI[1231] := 16#53E3;
   // UNI[1232] := 16#53E4;
   // UNI[1233] := 16#53E5;
   // UNI[1234] := 16#53E6;
   // UNI[1235] := 16#53E8;
   // UNI[1236] := 16#53E9;
   // UNI[1237] := 16#53EA;
   // UNI[1238] := 16#53EB;
   // UNI[1239] := 16#53EC;
   // UNI[1240] := 16#53ED;
   // UNI[1241] := 16#53EE;
   // UNI[1242] := 16#53EF;
   // UNI[1243] := 16#53F0;
   // UNI[1244] := 16#53F1;
   // UNI[1245] := 16#53F2;
   // UNI[1246] := 16#53F3;
   // UNI[1247] := 16#53F5;
   // UNI[1248] := 16#53F6;
   // UNI[1249] := 16#53F7;
   // UNI[1250] := 16#53F8;
   // UNI[1251] := 16#53F9;
   // UNI[1252] := 16#53FB;
   // UNI[1253] := 16#53FC;
   // UNI[1254] := 16#53FD;
   // UNI[1255] := 16#5401;
   // UNI[1256] := 16#5403;
   // UNI[1257] := 16#5404;
   // UNI[1258] := 16#5406;
   // UNI[1259] := 16#5408;
   // UNI[1260] := 16#5409;
   // UNI[1261] := 16#540A;
   // UNI[1262] := 16#540C;
   // UNI[1263] := 16#540D;
   // UNI[1264] := 16#540E;
   // UNI[1265] := 16#540F;
   // UNI[1266] := 16#5410;
   // UNI[1267] := 16#5411;
   // UNI[1268] := 16#5412;
   // UNI[1269] := 16#5413;
   // UNI[1270] := 16#5415;
   // UNI[1271] := 16#5416;
   // UNI[1272] := 16#5417;
   // UNI[1273] := 16#541B;
   // UNI[1274] := 16#541D;
   // UNI[1275] := 16#541E;
   // UNI[1276] := 16#541F;
   // UNI[1277] := 16#5420;
   // UNI[1278] := 16#5421;
   // UNI[1279] := 16#5423;
   // UNI[1280] := 16#5426;
   // UNI[1281] := 16#5427;
   // UNI[1282] := 16#5428;
   // UNI[1283] := 16#5429;
   // UNI[1284] := 16#542B;
   // UNI[1285] := 16#542C;
   // UNI[1286] := 16#542D;
   // UNI[1287] := 16#542E;
   // UNI[1288] := 16#542F;
   // UNI[1289] := 16#5431;
   // UNI[1290] := 16#5432;
   // UNI[1291] := 16#5434;
   // UNI[1292] := 16#5435;
   // UNI[1293] := 16#5438;
   // UNI[1294] := 16#5439;
   // UNI[1295] := 16#543B;
   // UNI[1296] := 16#543C;
   // UNI[1297] := 16#543E;
   // UNI[1298] := 16#5440;
   // UNI[1299] := 16#5443;
   // UNI[1300] := 16#5446;
   // UNI[1301] := 16#5448;
   // UNI[1302] := 16#544A;
   // UNI[1303] := 16#544B;
   // UNI[1304] := 16#5450;
   // UNI[1305] := 16#5452;
   // UNI[1306] := 16#5453;
   // UNI[1307] := 16#5454;
   // UNI[1308] := 16#5455;
   // UNI[1309] := 16#5456;
   // UNI[1310] := 16#5457;
   // UNI[1311] := 16#5458;
   // UNI[1312] := 16#5459;
   // UNI[1313] := 16#545B;
   // UNI[1314] := 16#545C;
   // UNI[1315] := 16#5462;
   // UNI[1316] := 16#5464;
   // UNI[1317] := 16#5466;
   // UNI[1318] := 16#5468;
   // UNI[1319] := 16#5471;
   // UNI[1320] := 16#5472;
   // UNI[1321] := 16#5473;
   // UNI[1322] := 16#5475;
   // UNI[1323] := 16#5476;
   // UNI[1324] := 16#5477;
   // UNI[1325] := 16#5478;
   // UNI[1326] := 16#547B;
   // UNI[1327] := 16#547C;
   // UNI[1328] := 16#547D;
   // UNI[1329] := 16#5480;
   // UNI[1330] := 16#5482;
   // UNI[1331] := 16#5484;
   // UNI[1332] := 16#5486;
   // UNI[1333] := 16#548B;
   // UNI[1334] := 16#548C;
   // UNI[1335] := 16#548E;
   // UNI[1336] := 16#548F;
   // UNI[1337] := 16#5490;
   // UNI[1338] := 16#5492;
   // UNI[1339] := 16#5494;
   // UNI[1340] := 16#5495;
   // UNI[1341] := 16#5496;
   // UNI[1342] := 16#5499;
   // UNI[1343] := 16#549A;
   // UNI[1344] := 16#549B;
   // UNI[1345] := 16#549D;
   // UNI[1346] := 16#54A3;
   // UNI[1347] := 16#54A4;
   // UNI[1348] := 16#54A6;
   // UNI[1349] := 16#54A7;
   // UNI[1350] := 16#54A8;
   // UNI[1351] := 16#54A9;
   // UNI[1352] := 16#54AA;
   // UNI[1353] := 16#54AB;
   // UNI[1354] := 16#54AC;
   // UNI[1355] := 16#54AD;
   // UNI[1356] := 16#54AF;
   // UNI[1357] := 16#54B1;
   // UNI[1358] := 16#54B3;
   // UNI[1359] := 16#54B4;
   // UNI[1360] := 16#54B8;
   // UNI[1361] := 16#54BB;
   // UNI[1362] := 16#54BD;
   // UNI[1363] := 16#54BF;
   // UNI[1364] := 16#54C0;
   // UNI[1365] := 16#54C1;
   // UNI[1366] := 16#54C2;
   // UNI[1367] := 16#54C4;
   // UNI[1368] := 16#54C6;
   // UNI[1369] := 16#54C7;
   // UNI[1370] := 16#54C8;
   // UNI[1371] := 16#54C9;
   // UNI[1372] := 16#54CC;
   // UNI[1373] := 16#54CD;
   // UNI[1374] := 16#54CE;
   // UNI[1375] := 16#54CF;
   // UNI[1376] := 16#54D0;
   // UNI[1377] := 16#54D1;
   // UNI[1378] := 16#54D2;
   // UNI[1379] := 16#54D3;
   // UNI[1380] := 16#54D4;
   // UNI[1381] := 16#54D5;
   // UNI[1382] := 16#54D7;
   // UNI[1383] := 16#54D9;
   // UNI[1384] := 16#54DA;
   // UNI[1385] := 16#54DC;
   // UNI[1386] := 16#54DD;
   // UNI[1387] := 16#54DE;
   // UNI[1388] := 16#54DF;
   // UNI[1389] := 16#54E5;
   // UNI[1390] := 16#54E6;
   // UNI[1391] := 16#54E7;
   // UNI[1392] := 16#54E8;
   // UNI[1393] := 16#54E9;
   // UNI[1394] := 16#54EA;
   // UNI[1395] := 16#54ED;
   // UNI[1396] := 16#54EE;
   // UNI[1397] := 16#54F2;
   // UNI[1398] := 16#54F3;
   // UNI[1399] := 16#54FA;
   // UNI[1400] := 16#54FC;
   // UNI[1401] := 16#54FD;
   // UNI[1402] := 16#54FF;
   // UNI[1403] := 16#5501;
   // UNI[1404] := 16#5506;
   // UNI[1405] := 16#5507;
   // UNI[1406] := 16#5509;
   // UNI[1407] := 16#550F;
   // UNI[1408] := 16#5510;
   // UNI[1409] := 16#5511;
   // UNI[1410] := 16#5514;
   // UNI[1411] := 16#551B;
   // UNI[1412] := 16#5520;
   // UNI[1413] := 16#5522;
   // UNI[1414] := 16#5523;
   // UNI[1415] := 16#5524;
   // UNI[1416] := 16#5527;
   // UNI[1417] := 16#552A;
   // UNI[1418] := 16#552C;
   // UNI[1419] := 16#552E;
   // UNI[1420] := 16#552F;
   // UNI[1421] := 16#5530;
   // UNI[1422] := 16#5531;
   // UNI[1423] := 16#5533;
   // UNI[1424] := 16#5537;
   // UNI[1425] := 16#553C;
   // UNI[1426] := 16#553E;
   // UNI[1427] := 16#553F;
   // UNI[1428] := 16#5541;
   // UNI[1429] := 16#5543;
   // UNI[1430] := 16#5544;
   // UNI[1431] := 16#5546;
   // UNI[1432] := 16#5549;
   // UNI[1433] := 16#554A;
   // UNI[1434] := 16#5550;
   // UNI[1435] := 16#5555;
   // UNI[1436] := 16#5556;
   // UNI[1437] := 16#555C;
   // UNI[1438] := 16#5561;
   // UNI[1439] := 16#5564;
   // UNI[1440] := 16#5565;
   // UNI[1441] := 16#5566;
   // UNI[1442] := 16#5567;
   // UNI[1443] := 16#556A;
   // UNI[1444] := 16#556C;
   // UNI[1445] := 16#556D;
   // UNI[1446] := 16#556E;
   // UNI[1447] := 16#5575;
   // UNI[1448] := 16#5576;
   // UNI[1449] := 16#5577;
   // UNI[1450] := 16#5578;
   // UNI[1451] := 16#557B;
   // UNI[1452] := 16#557C;
   // UNI[1453] := 16#557E;
   // UNI[1454] := 16#5580;
   // UNI[1455] := 16#5581;
   // UNI[1456] := 16#5582;
   // UNI[1457] := 16#5583;
   // UNI[1458] := 16#5584;
   // UNI[1459] := 16#5587;
   // UNI[1460] := 16#5588;
   // UNI[1461] := 16#5589;
   // UNI[1462] := 16#558A;
   // UNI[1463] := 16#558B;
   // UNI[1464] := 16#558F;
   // UNI[1465] := 16#5591;
   // UNI[1466] := 16#5594;
   // UNI[1467] := 16#5598;
   // UNI[1468] := 16#5599;
   // UNI[1469] := 16#559C;
   // UNI[1470] := 16#559D;
   // UNI[1471] := 16#559F;
   // UNI[1472] := 16#55A7;
   // UNI[1473] := 16#55B1;
   // UNI[1474] := 16#55B3;
   // UNI[1475] := 16#55B5;
   // UNI[1476] := 16#55B7;
   // UNI[1477] := 16#55B9;
   // UNI[1478] := 16#55BB;
   // UNI[1479] := 16#55BD;
   // UNI[1480] := 16#55BE;
   // UNI[1481] := 16#55C4;
   // UNI[1482] := 16#55C5;
   // UNI[1483] := 16#55C9;
   // UNI[1484] := 16#55CC;
   // UNI[1485] := 16#55CD;
   // UNI[1486] := 16#55D1;
   // UNI[1487] := 16#55D2;
   // UNI[1488] := 16#55D3;
   // UNI[1489] := 16#55D4;
   // UNI[1490] := 16#55D6;
   // UNI[1491] := 16#55DC;
   // UNI[1492] := 16#55DD;
   // UNI[1493] := 16#55DF;
   // UNI[1494] := 16#55E1;
   // UNI[1495] := 16#55E3;
   // UNI[1496] := 16#55E4;
   // UNI[1497] := 16#55E5;
   // UNI[1498] := 16#55E6;
   // UNI[1499] := 16#55E8;
   // UNI[1500] := 16#55EA;
   // UNI[1501] := 16#55EB;
   // UNI[1502] := 16#55EC;
   // UNI[1503] := 16#55EF;
   // UNI[1504] := 16#55F2;
   // UNI[1505] := 16#55F3;
   // UNI[1506] := 16#55F5;
   // UNI[1507] := 16#55F7;
   // UNI[1508] := 16#55FD;
   // UNI[1509] := 16#55FE;
   // UNI[1510] := 16#5600;
   // UNI[1511] := 16#5601;
   // UNI[1512] := 16#5608;
   // UNI[1513] := 16#5609;
   // UNI[1514] := 16#560C;
   // UNI[1515] := 16#560E;
   // UNI[1516] := 16#560F;
   // UNI[1517] := 16#5618;
   // UNI[1518] := 16#561B;
   // UNI[1519] := 16#561E;
   // UNI[1520] := 16#561F;
   // UNI[1521] := 16#5623;
   // UNI[1522] := 16#5624;
   // UNI[1523] := 16#5627;
   // UNI[1524] := 16#562C;
   // UNI[1525] := 16#562D;
   // UNI[1526] := 16#5631;
   // UNI[1527] := 16#5632;
   // UNI[1528] := 16#5634;
   // UNI[1529] := 16#5636;
   // UNI[1530] := 16#5639;
   // UNI[1531] := 16#563B;
   // UNI[1532] := 16#563F;
   // UNI[1533] := 16#564C;
   // UNI[1534] := 16#564D;
   // UNI[1535] := 16#564E;
   // UNI[1536] := 16#5654;
   // UNI[1537] := 16#5657;
   // UNI[1538] := 16#5658;
   // UNI[1539] := 16#5659;
   // UNI[1540] := 16#565C;
   // UNI[1541] := 16#5662;
   // UNI[1542] := 16#5664;
   // UNI[1543] := 16#5668;
   // UNI[1544] := 16#5669;
   // UNI[1545] := 16#566A;
   // UNI[1546] := 16#566B;
   // UNI[1547] := 16#566C;
   // UNI[1548] := 16#5671;
   // UNI[1549] := 16#5676;
   // UNI[1550] := 16#567B;
   // UNI[1551] := 16#567C;
   // UNI[1552] := 16#5685;
   // UNI[1553] := 16#5686;
   // UNI[1554] := 16#568E;
   // UNI[1555] := 16#568F;
   // UNI[1556] := 16#5693;
   // UNI[1557] := 16#56A3;
   // UNI[1558] := 16#56AF;
   // UNI[1559] := 16#56B7;
   // UNI[1560] := 16#56BC;
   // UNI[1561] := 16#56CA;
   // UNI[1562] := 16#56D4;
   // UNI[1563] := 16#56D7;
   // UNI[1564] := 16#56DA;
   // UNI[1565] := 16#56DB;
   // UNI[1566] := 16#56DD;
   // UNI[1567] := 16#56DE;
   // UNI[1568] := 16#56DF;
   // UNI[1569] := 16#56E0;
   // UNI[1570] := 16#56E1;
   // UNI[1571] := 16#56E2;
   // UNI[1572] := 16#56E4;
   // UNI[1573] := 16#56EB;
   // UNI[1574] := 16#56ED;
   // UNI[1575] := 16#56F0;
   // UNI[1576] := 16#56F1;
   // UNI[1577] := 16#56F4;
   // UNI[1578] := 16#56F5;
   // UNI[1579] := 16#56F9;
   // UNI[1580] := 16#56FA;
   // UNI[1581] := 16#56FD;
   // UNI[1582] := 16#56FE;
   // UNI[1583] := 16#56FF;
   // UNI[1584] := 16#5703;
   // UNI[1585] := 16#5704;
   // UNI[1586] := 16#5706;
   // UNI[1587] := 16#5708;
   // UNI[1588] := 16#5709;
   // UNI[1589] := 16#570A;
   // UNI[1590] := 16#571C;
   // UNI[1591] := 16#571F;
   // UNI[1592] := 16#5723;
   // UNI[1593] := 16#5728;
   // UNI[1594] := 16#5729;
   // UNI[1595] := 16#572A;
   // UNI[1596] := 16#572C;
   // UNI[1597] := 16#572D;
   // UNI[1598] := 16#572E;
   // UNI[1599] := 16#572F;
   // UNI[1600] := 16#5730;
   // UNI[1601] := 16#5733;
   // UNI[1602] := 16#5739;
   // UNI[1603] := 16#573A;
   // UNI[1604] := 16#573B;
   // UNI[1605] := 16#573E;
   // UNI[1606] := 16#5740;
   // UNI[1607] := 16#5742;
   // UNI[1608] := 16#5747;
   // UNI[1609] := 16#574A;
   // UNI[1610] := 16#574C;
   // UNI[1611] := 16#574D;
   // UNI[1612] := 16#574E;
   // UNI[1613] := 16#574F;
   // UNI[1614] := 16#5750;
   // UNI[1615] := 16#5751;
   // UNI[1616] := 16#5757;
   // UNI[1617] := 16#575A;
   // UNI[1618] := 16#575B;
   // UNI[1619] := 16#575C;
   // UNI[1620] := 16#575D;
   // UNI[1621] := 16#575E;
   // UNI[1622] := 16#575F;
   // UNI[1623] := 16#5760;
   // UNI[1624] := 16#5761;
   // UNI[1625] := 16#5764;
   // UNI[1626] := 16#5766;
   // UNI[1627] := 16#5768;
   // UNI[1628] := 16#5769;
   // UNI[1629] := 16#576A;
   // UNI[1630] := 16#576B;
   // UNI[1631] := 16#576D;
   // UNI[1632] := 16#576F;
   // UNI[1633] := 16#5773;
   // UNI[1634] := 16#5776;
   // UNI[1635] := 16#5777;
   // UNI[1636] := 16#577B;
   // UNI[1637] := 16#577C;
   // UNI[1638] := 16#5782;
   // UNI[1639] := 16#5783;
   // UNI[1640] := 16#5784;
   // UNI[1641] := 16#5785;
   // UNI[1642] := 16#5786;
   // UNI[1643] := 16#578B;
   // UNI[1644] := 16#578C;
   // UNI[1645] := 16#5792;
   // UNI[1646] := 16#5793;
   // UNI[1647] := 16#579B;
   // UNI[1648] := 16#57A0;
   // UNI[1649] := 16#57A1;
   // UNI[1650] := 16#57A2;
   // UNI[1651] := 16#57A3;
   // UNI[1652] := 16#57A4;
   // UNI[1653] := 16#57A6;
   // UNI[1654] := 16#57A7;
   // UNI[1655] := 16#57A9;
   // UNI[1656] := 16#57AB;
   // UNI[1657] := 16#57AD;
   // UNI[1658] := 16#57AE;
   // UNI[1659] := 16#57B2;
   // UNI[1660] := 16#57B4;
   // UNI[1661] := 16#57B8;
   // UNI[1662] := 16#57C2;
   // UNI[1663] := 16#57C3;
   // UNI[1664] := 16#57CB;
   // UNI[1665] := 16#57CE;
   // UNI[1666] := 16#57CF;
   // UNI[1667] := 16#57D2;
   // UNI[1668] := 16#57D4;
   // UNI[1669] := 16#57D5;
   // UNI[1670] := 16#57D8;
   // UNI[1671] := 16#57D9;
   // UNI[1672] := 16#57DA;
   // UNI[1673] := 16#57DD;
   // UNI[1674] := 16#57DF;
   // UNI[1675] := 16#57E0;
   // UNI[1676] := 16#57E4;
   // UNI[1677] := 16#57ED;
   // UNI[1678] := 16#57EF;
   // UNI[1679] := 16#57F4;
   // UNI[1680] := 16#57F8;
   // UNI[1681] := 16#57F9;
   // UNI[1682] := 16#57FA;
   // UNI[1683] := 16#57FD;
   // UNI[1684] := 16#5800;
   // UNI[1685] := 16#5802;
   // UNI[1686] := 16#5806;
   // UNI[1687] := 16#5807;
   // UNI[1688] := 16#580B;
   // UNI[1689] := 16#580D;
   // UNI[1690] := 16#5811;
   // UNI[1691] := 16#5815;
   // UNI[1692] := 16#5819;
   // UNI[1693] := 16#581E;
   // UNI[1694] := 16#5820;
   // UNI[1695] := 16#5821;
   // UNI[1696] := 16#5824;
   // UNI[1697] := 16#582A;
   // UNI[1698] := 16#5830;
   // UNI[1699] := 16#5835;
   // UNI[1700] := 16#5844;
   // UNI[1701] := 16#584C;
   // UNI[1702] := 16#584D;
   // UNI[1703] := 16#5851;
   // UNI[1704] := 16#5854;
   // UNI[1705] := 16#5858;
   // UNI[1706] := 16#585E;
   // UNI[1707] := 16#5865;
   // UNI[1708] := 16#586B;
   // UNI[1709] := 16#586C;
   // UNI[1710] := 16#587E;
   // UNI[1711] := 16#5880;
   // UNI[1712] := 16#5881;
   // UNI[1713] := 16#5883;
   // UNI[1714] := 16#5885;
   // UNI[1715] := 16#5889;
   // UNI[1716] := 16#5892;
   // UNI[1717] := 16#5893;
   // UNI[1718] := 16#5899;
   // UNI[1719] := 16#589A;
   // UNI[1720] := 16#589E;
   // UNI[1721] := 16#589F;
   // UNI[1722] := 16#58A8;
   // UNI[1723] := 16#58A9;
   // UNI[1724] := 16#58BC;
   // UNI[1725] := 16#58C1;
   // UNI[1726] := 16#58C5;
   // UNI[1727] := 16#58D1;
   // UNI[1728] := 16#58D5;
   // UNI[1729] := 16#58E4;
   // UNI[1730] := 16#58EB;
   // UNI[1731] := 16#58EC;
   // UNI[1732] := 16#58EE;
   // UNI[1733] := 16#58F0;
   // UNI[1734] := 16#58F3;
   // UNI[1735] := 16#58F6;
   // UNI[1736] := 16#58F9;
   // UNI[1737] := 16#5902;
   // UNI[1738] := 16#5904;
   // UNI[1739] := 16#5907;
   // UNI[1740] := 16#590D;
   // UNI[1741] := 16#590F;
   // UNI[1742] := 16#5914;
   // UNI[1743] := 16#5915;
   // UNI[1744] := 16#5916;
   // UNI[1745] := 16#5919;
   // UNI[1746] := 16#591A;
   // UNI[1747] := 16#591C;
   // UNI[1748] := 16#591F;
   // UNI[1749] := 16#5924;
   // UNI[1750] := 16#5925;
   // UNI[1751] := 16#5927;
   // UNI[1752] := 16#5929;
   // UNI[1753] := 16#592A;
   // UNI[1754] := 16#592B;
   // UNI[1755] := 16#592D;
   // UNI[1756] := 16#592E;
   // UNI[1757] := 16#592F;
   // UNI[1758] := 16#5931;
   // UNI[1759] := 16#5934;
   // UNI[1760] := 16#5937;
   // UNI[1761] := 16#5938;
   // UNI[1762] := 16#5939;
   // UNI[1763] := 16#593A;
   // UNI[1764] := 16#593C;
   // UNI[1765] := 16#5941;
   // UNI[1766] := 16#5942;
   // UNI[1767] := 16#5944;
   // UNI[1768] := 16#5947;
   // UNI[1769] := 16#5948;
   // UNI[1770] := 16#5949;
   // UNI[1771] := 16#594B;
   // UNI[1772] := 16#594E;
   // UNI[1773] := 16#594F;
   // UNI[1774] := 16#5951;
   // UNI[1775] := 16#5954;
   // UNI[1776] := 16#5955;
   // UNI[1777] := 16#5956;
   // UNI[1778] := 16#5957;
   // UNI[1779] := 16#5958;
   // UNI[1780] := 16#595A;
   // UNI[1781] := 16#5960;
   // UNI[1782] := 16#5962;
   // UNI[1783] := 16#5965;
   // UNI[1784] := 16#5973;
   // UNI[1785] := 16#5974;
   // UNI[1786] := 16#5976;
   // UNI[1787] := 16#5978;
   // UNI[1788] := 16#5979;
   // UNI[1789] := 16#597D;
   // UNI[1790] := 16#5981;
   // UNI[1791] := 16#5982;
   // UNI[1792] := 16#5983;
   // UNI[1793] := 16#5984;
   // UNI[1794] := 16#5986;
   // UNI[1795] := 16#5987;
   // UNI[1796] := 16#5988;
   // UNI[1797] := 16#598A;
   // UNI[1798] := 16#598D;
   // UNI[1799] := 16#5992;
   // UNI[1800] := 16#5993;
   // UNI[1801] := 16#5996;
   // UNI[1802] := 16#5997;
   // UNI[1803] := 16#5999;
   // UNI[1804] := 16#599E;
   // UNI[1805] := 16#59A3;
   // UNI[1806] := 16#59A4;
   // UNI[1807] := 16#59A5;
   // UNI[1808] := 16#59A8;
   // UNI[1809] := 16#59A9;
   // UNI[1810] := 16#59AA;
   // UNI[1811] := 16#59AB;
   // UNI[1812] := 16#59AE;
   // UNI[1813] := 16#59AF;
   // UNI[1814] := 16#59B2;
   // UNI[1815] := 16#59B9;
   // UNI[1816] := 16#59BB;
   // UNI[1817] := 16#59BE;
   // UNI[1818] := 16#59C6;
   // UNI[1819] := 16#59CA;
   // UNI[1820] := 16#59CB;
   // UNI[1821] := 16#59D0;
   // UNI[1822] := 16#59D1;
   // UNI[1823] := 16#59D2;
   // UNI[1824] := 16#59D3;
   // UNI[1825] := 16#59D4;
   // UNI[1826] := 16#59D7;
   // UNI[1827] := 16#59D8;
   // UNI[1828] := 16#59DA;
   // UNI[1829] := 16#59DC;
   // UNI[1830] := 16#59DD;
   // UNI[1831] := 16#59E3;
   // UNI[1832] := 16#59E5;
   // UNI[1833] := 16#59E8;
   // UNI[1834] := 16#59EC;
   // UNI[1835] := 16#59F9;
   // UNI[1836] := 16#59FB;
   // UNI[1837] := 16#59FF;
   // UNI[1838] := 16#5A01;
   // UNI[1839] := 16#5A03;
   // UNI[1840] := 16#5A04;
   // UNI[1841] := 16#5A05;
   // UNI[1842] := 16#5A06;
   // UNI[1843] := 16#5A07;
   // UNI[1844] := 16#5A08;
   // UNI[1845] := 16#5A09;
   // UNI[1846] := 16#5A0C;
   // UNI[1847] := 16#5A11;
   // UNI[1848] := 16#5A13;
   // UNI[1849] := 16#5A18;
   // UNI[1850] := 16#5A1C;
   // UNI[1851] := 16#5A1F;
   // UNI[1852] := 16#5A20;
   // UNI[1853] := 16#5A23;
   // UNI[1854] := 16#5A25;
   // UNI[1855] := 16#5A29;
   // UNI[1856] := 16#5A31;
   // UNI[1857] := 16#5A32;
   // UNI[1858] := 16#5A34;
   // UNI[1859] := 16#5A36;
   // UNI[1860] := 16#5A3C;
   // UNI[1861] := 16#5A40;
   // UNI[1862] := 16#5A46;
   // UNI[1863] := 16#5A49;
   // UNI[1864] := 16#5A4A;
   // UNI[1865] := 16#5A55;
   // UNI[1866] := 16#5A5A;
   // UNI[1867] := 16#5A62;
   // UNI[1868] := 16#5A67;
   // UNI[1869] := 16#5A6A;
   // UNI[1870] := 16#5A74;
   // UNI[1871] := 16#5A75;
   // UNI[1872] := 16#5A76;
   // UNI[1873] := 16#5A77;
   // UNI[1874] := 16#5A7A;
   // UNI[1875] := 16#5A7F;
   // UNI[1876] := 16#5A92;
   // UNI[1877] := 16#5A9A;
   // UNI[1878] := 16#5A9B;
   // UNI[1879] := 16#5AAA;
   // UNI[1880] := 16#5AB2;
   // UNI[1881] := 16#5AB3;
   // UNI[1882] := 16#5AB5;
   // UNI[1883] := 16#5AB8;
   // UNI[1884] := 16#5ABE;
   // UNI[1885] := 16#5AC1;
   // UNI[1886] := 16#5AC2;
   // UNI[1887] := 16#5AC9;
   // UNI[1888] := 16#5ACC;
   // UNI[1889] := 16#5AD2;
   // UNI[1890] := 16#5AD4;
   // UNI[1891] := 16#5AD6;
   // UNI[1892] := 16#5AD8;
   // UNI[1893] := 16#5ADC;
   // UNI[1894] := 16#5AE0;
   // UNI[1895] := 16#5AE1;
   // UNI[1896] := 16#5AE3;
   // UNI[1897] := 16#5AE6;
   // UNI[1898] := 16#5AE9;
   // UNI[1899] := 16#5AEB;
   // UNI[1900] := 16#5AF1;
   // UNI[1901] := 16#5B09;
   // UNI[1902] := 16#5B16;
   // UNI[1903] := 16#5B17;
   // UNI[1904] := 16#5B32;
   // UNI[1905] := 16#5B34;
   // UNI[1906] := 16#5B37;
   // UNI[1907] := 16#5B40;
   // UNI[1908] := 16#5B50;
   // UNI[1909] := 16#5B51;
   // UNI[1910] := 16#5B53;
   // UNI[1911] := 16#5B54;
   // UNI[1912] := 16#5B55;
   // UNI[1913] := 16#5B57;
   // UNI[1914] := 16#5B58;
   // UNI[1915] := 16#5B59;
   // UNI[1916] := 16#5B5A;
   // UNI[1917] := 16#5B5B;
   // UNI[1918] := 16#5B5C;
   // UNI[1919] := 16#5B5D;
   // UNI[1920] := 16#5B5F;
   // UNI[1921] := 16#5B62;
   // UNI[1922] := 16#5B63;
   // UNI[1923] := 16#5B64;
   // UNI[1924] := 16#5B65;
   // UNI[1925] := 16#5B66;
   // UNI[1926] := 16#5B69;
   // UNI[1927] := 16#5B6A;
   // UNI[1928] := 16#5B6C;
   // UNI[1929] := 16#5B70;
   // UNI[1930] := 16#5B71;
   // UNI[1931] := 16#5B73;
   // UNI[1932] := 16#5B75;
   // UNI[1933] := 16#5B7A;
   // UNI[1934] := 16#5B7D;
   // UNI[1935] := 16#5B80;
   // UNI[1936] := 16#5B81;
   // UNI[1937] := 16#5B83;
   // UNI[1938] := 16#5B84;
   // UNI[1939] := 16#5B85;
   // UNI[1940] := 16#5B87;
   // UNI[1941] := 16#5B88;
   // UNI[1942] := 16#5B89;
   // UNI[1943] := 16#5B8B;
   // UNI[1944] := 16#5B8C;
   // UNI[1945] := 16#5B8F;
   // UNI[1946] := 16#5B93;
   // UNI[1947] := 16#5B95;
   // UNI[1948] := 16#5B97;
   // UNI[1949] := 16#5B98;
   // UNI[1950] := 16#5B99;
   // UNI[1951] := 16#5B9A;
   // UNI[1952] := 16#5B9B;
   // UNI[1953] := 16#5B9C;
   // UNI[1954] := 16#5B9D;
   // UNI[1955] := 16#5B9E;
   // UNI[1956] := 16#5BA0;
   // UNI[1957] := 16#5BA1;
   // UNI[1958] := 16#5BA2;
   // UNI[1959] := 16#5BA3;
   // UNI[1960] := 16#5BA4;
   // UNI[1961] := 16#5BA5;
   // UNI[1962] := 16#5BA6;
   // UNI[1963] := 16#5BAA;
   // UNI[1964] := 16#5BAB;
   // UNI[1965] := 16#5BB0;
   // UNI[1966] := 16#5BB3;
   // UNI[1967] := 16#5BB4;
   // UNI[1968] := 16#5BB5;
   // UNI[1969] := 16#5BB6;
   // UNI[1970] := 16#5BB8;
   // UNI[1971] := 16#5BB9;
   // UNI[1972] := 16#5BBD;
   // UNI[1973] := 16#5BBE;
   // UNI[1974] := 16#5BBF;
   // UNI[1975] := 16#5BC2;
   // UNI[1976] := 16#5BC4;
   // UNI[1977] := 16#5BC5;
   // UNI[1978] := 16#5BC6;
   // UNI[1979] := 16#5BC7;
   // UNI[1980] := 16#5BCC;
   // UNI[1981] := 16#5BD0;
   // UNI[1982] := 16#5BD2;
   // UNI[1983] := 16#5BD3;
   // UNI[1984] := 16#5BDD;
   // UNI[1985] := 16#5BDE;
   // UNI[1986] := 16#5BDF;
   // UNI[1987] := 16#5BE1;
   // UNI[1988] := 16#5BE4;
   // UNI[1989] := 16#5BE5;
   // UNI[1990] := 16#5BE8;
   // UNI[1991] := 16#5BEE;
   // UNI[1992] := 16#5BF0;
   // UNI[1993] := 16#5BF8;
   // UNI[1994] := 16#5BF9;
   // UNI[1995] := 16#5BFA;
   // UNI[1996] := 16#5BFB;
   // UNI[1997] := 16#5BFC;
   // UNI[1998] := 16#5BFF;
   // UNI[1999] := 16#5C01;
   // UNI[2000] := 16#5C04;
   // UNI[2001] := 16#5C06;
   // UNI[2002] := 16#5C09;
   // UNI[2003] := 16#5C0A;
   // UNI[2004] := 16#5C0F;
   // UNI[2005] := 16#5C11;
   // UNI[2006] := 16#5C14;
   // UNI[2007] := 16#5C15;
   // UNI[2008] := 16#5C16;
   // UNI[2009] := 16#5C18;
   // UNI[2010] := 16#5C1A;
   // UNI[2011] := 16#5C1C;
   // UNI[2012] := 16#5C1D;
   // UNI[2013] := 16#5C22;
   // UNI[2014] := 16#5C24;
   // UNI[2015] := 16#5C25;
   // UNI[2016] := 16#5C27;
   // UNI[2017] := 16#5C2C;
   // UNI[2018] := 16#5C31;
   // UNI[2019] := 16#5C34;
   // UNI[2020] := 16#5C38;
   // UNI[2021] := 16#5C39;
   // UNI[2022] := 16#5C3A;
   // UNI[2023] := 16#5C3B;
   // UNI[2024] := 16#5C3C;
   // UNI[2025] := 16#5C3D;
   // UNI[2026] := 16#5C3E;
   // UNI[2027] := 16#5C3F;
   // UNI[2028] := 16#5C40;
   // UNI[2029] := 16#5C41;
   // UNI[2030] := 16#5C42;
   // UNI[2031] := 16#5C45;
   // UNI[2032] := 16#5C48;
   // UNI[2033] := 16#5C49;
   // UNI[2034] := 16#5C4A;
   // UNI[2035] := 16#5C4B;
   // UNI[2036] := 16#5C4E;
   // UNI[2037] := 16#5C4F;
   // UNI[2038] := 16#5C50;
   // UNI[2039] := 16#5C51;
   // UNI[2040] := 16#5C55;
   // UNI[2041] := 16#5C59;
   // UNI[2042] := 16#5C5E;
   // UNI[2043] := 16#5C60;
   // UNI[2044] := 16#5C61;
   // UNI[2045] := 16#5C63;
   // UNI[2046] := 16#5C65;
   // UNI[2047] := 16#5C66;
   // UNI[2048] := 16#5C6E;
   // UNI[2049] := 16#5C6F;
   // UNI[2050] := 16#5C71;
   // UNI[2051] := 16#5C79;
   // UNI[2052] := 16#5C7A;
   // UNI[2053] := 16#5C7F;
   // UNI[2054] := 16#5C81;
   // UNI[2055] := 16#5C82;
   // UNI[2056] := 16#5C88;
   // UNI[2057] := 16#5C8C;
   // UNI[2058] := 16#5C8D;
   // UNI[2059] := 16#5C90;
   // UNI[2060] := 16#5C91;
   // UNI[2061] := 16#5C94;
   // UNI[2062] := 16#5C96;
   // UNI[2063] := 16#5C97;
   // UNI[2064] := 16#5C98;
   // UNI[2065] := 16#5C99;
   // UNI[2066] := 16#5C9A;
   // UNI[2067] := 16#5C9B;
   // UNI[2068] := 16#5C9C;
   // UNI[2069] := 16#5CA2;
   // UNI[2070] := 16#5CA3;
   // UNI[2071] := 16#5CA9;
   // UNI[2072] := 16#5CAB;
   // UNI[2073] := 16#5CAC;
   // UNI[2074] := 16#5CAD;
   // UNI[2075] := 16#5CB1;
   // UNI[2076] := 16#5CB3;
   // UNI[2077] := 16#5CB5;
   // UNI[2078] := 16#5CB7;
   // UNI[2079] := 16#5CB8;
   // UNI[2080] := 16#5CBD;
   // UNI[2081] := 16#5CBF;
   // UNI[2082] := 16#5CC1;
   // UNI[2083] := 16#5CC4;
   // UNI[2084] := 16#5CCB;
   // UNI[2085] := 16#5CD2;
   // UNI[2086] := 16#5CD9;
   // UNI[2087] := 16#5CE1;
   // UNI[2088] := 16#5CE4;
   // UNI[2089] := 16#5CE5;
   // UNI[2090] := 16#5CE6;
   // UNI[2091] := 16#5CE8;
   // UNI[2092] := 16#5CEA;
   // UNI[2093] := 16#5CED;
   // UNI[2094] := 16#5CF0;
   // UNI[2095] := 16#5CFB;
   // UNI[2096] := 16#5D02;
   // UNI[2097] := 16#5D03;
   // UNI[2098] := 16#5D06;
   // UNI[2099] := 16#5D07;
   // UNI[2100] := 16#5D0E;
   // UNI[2101] := 16#5D14;
   // UNI[2102] := 16#5D16;
   // UNI[2103] := 16#5D1B;
   // UNI[2104] := 16#5D1E;
   // UNI[2105] := 16#5D24;
   // UNI[2106] := 16#5D26;
   // UNI[2107] := 16#5D27;
   // UNI[2108] := 16#5D29;
   // UNI[2109] := 16#5D2D;
   // UNI[2110] := 16#5D2E;
   // UNI[2111] := 16#5D34;
   // UNI[2112] := 16#5D3D;
   // UNI[2113] := 16#5D3E;
   // UNI[2114] := 16#5D47;
   // UNI[2115] := 16#5D4A;
   // UNI[2116] := 16#5D4B;
   // UNI[2117] := 16#5D4C;
   // UNI[2118] := 16#5D58;
   // UNI[2119] := 16#5D5B;
   // UNI[2120] := 16#5D5D;
   // UNI[2121] := 16#5D69;
   // UNI[2122] := 16#5D6B;
   // UNI[2123] := 16#5D6C;
   // UNI[2124] := 16#5D6F;
   // UNI[2125] := 16#5D74;
   // UNI[2126] := 16#5D82;
   // UNI[2127] := 16#5D99;
   // UNI[2128] := 16#5D9D;
   // UNI[2129] := 16#5DB7;
   // UNI[2130] := 16#5DC5;
   // UNI[2131] := 16#5DCD;
   // UNI[2132] := 16#5DDB;
   // UNI[2133] := 16#5DDD;
   // UNI[2134] := 16#5DDE;
   // UNI[2135] := 16#5DE1;
   // UNI[2136] := 16#5DE2;
   // UNI[2137] := 16#5DE5;
   // UNI[2138] := 16#5DE6;
   // UNI[2139] := 16#5DE7;
   // UNI[2140] := 16#5DE8;
   // UNI[2141] := 16#5DE9;
   // UNI[2142] := 16#5DEB;
   // UNI[2143] := 16#5DEE;
   // UNI[2144] := 16#5DEF;
   // UNI[2145] := 16#5DF1;
   // UNI[2146] := 16#5DF2;
   // UNI[2147] := 16#5DF3;
   // UNI[2148] := 16#5DF4;
   // UNI[2149] := 16#5DF7;
   // UNI[2150] := 16#5DFD;
   // UNI[2151] := 16#5DFE;
   // UNI[2152] := 16#5E01;
   // UNI[2153] := 16#5E02;
   // UNI[2154] := 16#5E03;
   // UNI[2155] := 16#5E05;
   // UNI[2156] := 16#5E06;
   // UNI[2157] := 16#5E08;
   // UNI[2158] := 16#5E0C;
   // UNI[2159] := 16#5E0F;
   // UNI[2160] := 16#5E10;
   // UNI[2161] := 16#5E11;
   // UNI[2162] := 16#5E14;
   // UNI[2163] := 16#5E15;
   // UNI[2164] := 16#5E16;
   // UNI[2165] := 16#5E18;
   // UNI[2166] := 16#5E19;
   // UNI[2167] := 16#5E1A;
   // UNI[2168] := 16#5E1B;
   // UNI[2169] := 16#5E1C;
   // UNI[2170] := 16#5E1D;
   // UNI[2171] := 16#5E26;
   // UNI[2172] := 16#5E27;
   // UNI[2173] := 16#5E2D;
   // UNI[2174] := 16#5E2E;
   // UNI[2175] := 16#5E31;
   // UNI[2176] := 16#5E37;
   // UNI[2177] := 16#5E38;
   // UNI[2178] := 16#5E3B;
   // UNI[2179] := 16#5E3C;
   // UNI[2180] := 16#5E3D;
   // UNI[2181] := 16#5E42;
   // UNI[2182] := 16#5E44;
   // UNI[2183] := 16#5E45;
   // UNI[2184] := 16#5E4C;
   // UNI[2185] := 16#5E54;
   // UNI[2186] := 16#5E55;
   // UNI[2187] := 16#5E5B;
   // UNI[2188] := 16#5E5E;
   // UNI[2189] := 16#5E61;
   // UNI[2190] := 16#5E62;
   // UNI[2191] := 16#5E72;
   // UNI[2192] := 16#5E73;
   // UNI[2193] := 16#5E74;
   // UNI[2194] := 16#5E76;
   // UNI[2195] := 16#5E78;
   // UNI[2196] := 16#5E7A;
   // UNI[2197] := 16#5E7B;
   // UNI[2198] := 16#5E7C;
   // UNI[2199] := 16#5E7D;
   // UNI[2200] := 16#5E7F;
   // UNI[2201] := 16#5E80;
   // UNI[2202] := 16#5E84;
   // UNI[2203] := 16#5E86;
   // UNI[2204] := 16#5E87;
   // UNI[2205] := 16#5E8A;
   // UNI[2206] := 16#5E8B;
   // UNI[2207] := 16#5E8F;
   // UNI[2208] := 16#5E90;
   // UNI[2209] := 16#5E91;
   // UNI[2210] := 16#5E93;
   // UNI[2211] := 16#5E94;
   // UNI[2212] := 16#5E95;
   // UNI[2213] := 16#5E96;
   // UNI[2214] := 16#5E97;
   // UNI[2215] := 16#5E99;
   // UNI[2216] := 16#5E9A;
   // UNI[2217] := 16#5E9C;
   // UNI[2218] := 16#5E9E;
   // UNI[2219] := 16#5E9F;
   // UNI[2220] := 16#5EA0;
   // UNI[2221] := 16#5EA5;
   // UNI[2222] := 16#5EA6;
   // UNI[2223] := 16#5EA7;
   // UNI[2224] := 16#5EAD;
   // UNI[2225] := 16#5EB3;
   // UNI[2226] := 16#5EB5;
   // UNI[2227] := 16#5EB6;
   // UNI[2228] := 16#5EB7;
   // UNI[2229] := 16#5EB8;
   // UNI[2230] := 16#5EB9;
   // UNI[2231] := 16#5EBE;
   // UNI[2232] := 16#5EC9;
   // UNI[2233] := 16#5ECA;
   // UNI[2234] := 16#5ED1;
   // UNI[2235] := 16#5ED2;
   // UNI[2236] := 16#5ED3;
   // UNI[2237] := 16#5ED6;
   // UNI[2238] := 16#5EDB;
   // UNI[2239] := 16#5EE8;
   // UNI[2240] := 16#5EEA;
   // UNI[2241] := 16#5EF4;
   // UNI[2242] := 16#5EF6;
   // UNI[2243] := 16#5EF7;
   // UNI[2244] := 16#5EFA;
   // UNI[2245] := 16#5EFE;
   // UNI[2246] := 16#5EFF;
   // UNI[2247] := 16#5F00;
   // UNI[2248] := 16#5F01;
   // UNI[2249] := 16#5F02;
   // UNI[2250] := 16#5F03;
   // UNI[2251] := 16#5F04;
   // UNI[2252] := 16#5F08;
   // UNI[2253] := 16#5F0A;
   // UNI[2254] := 16#5F0B;
   // UNI[2255] := 16#5F0F;
   // UNI[2256] := 16#5F11;
   // UNI[2257] := 16#5F13;
   // UNI[2258] := 16#5F15;
   // UNI[2259] := 16#5F17;
   // UNI[2260] := 16#5F18;
   // UNI[2261] := 16#5F1B;
   // UNI[2262] := 16#5F1F;
   // UNI[2263] := 16#5F20;
   // UNI[2264] := 16#5F25;
   // UNI[2265] := 16#5F26;
   // UNI[2266] := 16#5F27;
   // UNI[2267] := 16#5F29;
   // UNI[2268] := 16#5F2A;
   // UNI[2269] := 16#5F2D;
   // UNI[2270] := 16#5F2F;
   // UNI[2271] := 16#5F31;
   // UNI[2272] := 16#5F39;
   // UNI[2273] := 16#5F3A;
   // UNI[2274] := 16#5F3C;
   // UNI[2275] := 16#5F40;
   // UNI[2276] := 16#5F50;
   // UNI[2277] := 16#5F52;
   // UNI[2278] := 16#5F53;
   // UNI[2279] := 16#5F55;
   // UNI[2280] := 16#5F56;
   // UNI[2281] := 16#5F57;
   // UNI[2282] := 16#5F58;
   // UNI[2283] := 16#5F5D;
   // UNI[2284] := 16#5F61;
   // UNI[2285] := 16#5F62;
   // UNI[2286] := 16#5F64;
   // UNI[2287] := 16#5F66;
   // UNI[2288] := 16#5F69;
   // UNI[2289] := 16#5F6A;
   // UNI[2290] := 16#5F6C;
   // UNI[2291] := 16#5F6D;
   // UNI[2292] := 16#5F70;
   // UNI[2293] := 16#5F71;
   // UNI[2294] := 16#5F73;
   // UNI[2295] := 16#5F77;
   // UNI[2296] := 16#5F79;
   // UNI[2297] := 16#5F7B;
   // UNI[2298] := 16#5F7C;
   // UNI[2299] := 16#5F80;
   // UNI[2300] := 16#5F81;
   // UNI[2301] := 16#5F82;
   // UNI[2302] := 16#5F84;
   // UNI[2303] := 16#5F85;
   // UNI[2304] := 16#5F87;
   // UNI[2305] := 16#5F88;
   // UNI[2306] := 16#5F89;
   // UNI[2307] := 16#5F8A;
   // UNI[2308] := 16#5F8B;
   // UNI[2309] := 16#5F8C;
   // UNI[2310] := 16#5F90;
   // UNI[2311] := 16#5F92;
   // UNI[2312] := 16#5F95;
   // UNI[2313] := 16#5F97;
   // UNI[2314] := 16#5F98;
   // UNI[2315] := 16#5F99;
   // UNI[2316] := 16#5F9C;
   // UNI[2317] := 16#5FA1;
   // UNI[2318] := 16#5FA8;
   // UNI[2319] := 16#5FAA;
   // UNI[2320] := 16#5FAD;
   // UNI[2321] := 16#5FAE;
   // UNI[2322] := 16#5FB5;
   // UNI[2323] := 16#5FB7;
   // UNI[2324] := 16#5FBC;
   // UNI[2325] := 16#5FBD;
   // UNI[2326] := 16#5FC3;
   // UNI[2327] := 16#5FC4;
   // UNI[2328] := 16#5FC5;
   // UNI[2329] := 16#5FC6;
   // UNI[2330] := 16#5FC9;
   // UNI[2331] := 16#5FCC;
   // UNI[2332] := 16#5FCD;
   // UNI[2333] := 16#5FCF;
   // UNI[2334] := 16#5FD0;
   // UNI[2335] := 16#5FD1;
   // UNI[2336] := 16#5FD2;
   // UNI[2337] := 16#5FD6;
   // UNI[2338] := 16#5FD7;
   // UNI[2339] := 16#5FD8;
   // UNI[2340] := 16#5FD9;
   // UNI[2341] := 16#5FDD;
   // UNI[2342] := 16#5FE0;
   // UNI[2343] := 16#5FE1;
   // UNI[2344] := 16#5FE4;
   // UNI[2345] := 16#5FE7;
   // UNI[2346] := 16#5FEA;
   // UNI[2347] := 16#5FEB;
   // UNI[2348] := 16#5FED;
   // UNI[2349] := 16#5FEE;
   // UNI[2350] := 16#5FF1;
   // UNI[2351] := 16#5FF5;
   // UNI[2352] := 16#5FF8;
   // UNI[2353] := 16#5FFB;
   // UNI[2354] := 16#5FFD;
   // UNI[2355] := 16#5FFE;
   // UNI[2356] := 16#5FFF;
   // UNI[2357] := 16#6000;
   // UNI[2358] := 16#6001;
   // UNI[2359] := 16#6002;
   // UNI[2360] := 16#6003;
   // UNI[2361] := 16#6004;
   // UNI[2362] := 16#6005;
   // UNI[2363] := 16#6006;
   // UNI[2364] := 16#600A;
   // UNI[2365] := 16#600D;
   // UNI[2366] := 16#600E;
   // UNI[2367] := 16#600F;
   // UNI[2368] := 16#6012;
   // UNI[2369] := 16#6014;
   // UNI[2370] := 16#6015;
   // UNI[2371] := 16#6016;
   // UNI[2372] := 16#6019;
   // UNI[2373] := 16#601B;
   // UNI[2374] := 16#601C;
   // UNI[2375] := 16#601D;
   // UNI[2376] := 16#6020;
   // UNI[2377] := 16#6021;
   // UNI[2378] := 16#6025;
   // UNI[2379] := 16#6026;
   // UNI[2380] := 16#6027;
   // UNI[2381] := 16#6028;
   // UNI[2382] := 16#6029;
   // UNI[2383] := 16#602A;
   // UNI[2384] := 16#602B;
   // UNI[2385] := 16#602F;
   // UNI[2386] := 16#6035;
   // UNI[2387] := 16#603B;
   // UNI[2388] := 16#603C;
   // UNI[2389] := 16#603F;
   // UNI[2390] := 16#6041;
   // UNI[2391] := 16#6042;
   // UNI[2392] := 16#6043;
   // UNI[2393] := 16#604B;
   // UNI[2394] := 16#604D;
   // UNI[2395] := 16#6050;
   // UNI[2396] := 16#6052;
   // UNI[2397] := 16#6055;
   // UNI[2398] := 16#6059;
   // UNI[2399] := 16#605A;
   // UNI[2400] := 16#605D;
   // UNI[2401] := 16#6062;
   // UNI[2402] := 16#6063;
   // UNI[2403] := 16#6064;
   // UNI[2404] := 16#6067;
   // UNI[2405] := 16#6068;
   // UNI[2406] := 16#6069;
   // UNI[2407] := 16#606A;
   // UNI[2408] := 16#606B;
   // UNI[2409] := 16#606C;
   // UNI[2410] := 16#606D;
   // UNI[2411] := 16#606F;
   // UNI[2412] := 16#6070;
   // UNI[2413] := 16#6073;
   // UNI[2414] := 16#6076;
   // UNI[2415] := 16#6078;
   // UNI[2416] := 16#6079;
   // UNI[2417] := 16#607A;
   // UNI[2418] := 16#607B;
   // UNI[2419] := 16#607C;
   // UNI[2420] := 16#607D;
   // UNI[2421] := 16#607F;
   // UNI[2422] := 16#6083;
   // UNI[2423] := 16#6084;
   // UNI[2424] := 16#6089;
   // UNI[2425] := 16#608C;
   // UNI[2426] := 16#608D;
   // UNI[2427] := 16#6092;
   // UNI[2428] := 16#6094;
   // UNI[2429] := 16#6096;
   // UNI[2430] := 16#609A;
   // UNI[2431] := 16#609B;
   // UNI[2432] := 16#609D;
   // UNI[2433] := 16#609F;
   // UNI[2434] := 16#60A0;
   // UNI[2435] := 16#60A3;
   // UNI[2436] := 16#60A6;
   // UNI[2437] := 16#60A8;
   // UNI[2438] := 16#60AB;
   // UNI[2439] := 16#60AC;
   // UNI[2440] := 16#60AD;
   // UNI[2441] := 16#60AF;
   // UNI[2442] := 16#60B1;
   // UNI[2443] := 16#60B2;
   // UNI[2444] := 16#60B4;
   // UNI[2445] := 16#60B8;
   // UNI[2446] := 16#60BB;
   // UNI[2447] := 16#60BC;
   // UNI[2448] := 16#60C5;
   // UNI[2449] := 16#60C6;
   // UNI[2450] := 16#60CA;
   // UNI[2451] := 16#60CB;
   // UNI[2452] := 16#60D1;
   // UNI[2453] := 16#60D5;
   // UNI[2454] := 16#60D8;
   // UNI[2455] := 16#60DA;
   // UNI[2456] := 16#60DC;
   // UNI[2457] := 16#60DD;
   // UNI[2458] := 16#60DF;
   // UNI[2459] := 16#60E0;
   // UNI[2460] := 16#60E6;
   // UNI[2461] := 16#60E7;
   // UNI[2462] := 16#60E8;
   // UNI[2463] := 16#60E9;
   // UNI[2464] := 16#60EB;
   // UNI[2465] := 16#60EC;
   // UNI[2466] := 16#60ED;
   // UNI[2467] := 16#60EE;
   // UNI[2468] := 16#60EF;
   // UNI[2469] := 16#60F0;
   // UNI[2470] := 16#60F3;
   // UNI[2471] := 16#60F4;
   // UNI[2472] := 16#60F6;
   // UNI[2473] := 16#60F9;
   // UNI[2474] := 16#60FA;
   // UNI[2475] := 16#6100;
   // UNI[2476] := 16#6101;
   // UNI[2477] := 16#6106;
   // UNI[2478] := 16#6108;
   // UNI[2479] := 16#6109;
   // UNI[2480] := 16#610D;
   // UNI[2481] := 16#610E;
   // UNI[2482] := 16#610F;
   // UNI[2483] := 16#6115;
   // UNI[2484] := 16#611A;
   // UNI[2485] := 16#611F;
   // UNI[2486] := 16#6120;
   // UNI[2487] := 16#6123;
   // UNI[2488] := 16#6124;
   // UNI[2489] := 16#6126;
   // UNI[2490] := 16#6127;
   // UNI[2491] := 16#612B;
   // UNI[2492] := 16#613F;
   // UNI[2493] := 16#6148;
   // UNI[2494] := 16#614A;
   // UNI[2495] := 16#614C;
   // UNI[2496] := 16#614E;
   // UNI[2497] := 16#6151;
   // UNI[2498] := 16#6155;
   // UNI[2499] := 16#615D;
   // UNI[2500] := 16#6162;
   // UNI[2501] := 16#6167;
   // UNI[2502] := 16#6168;
   // UNI[2503] := 16#6170;
   // UNI[2504] := 16#6175;
   // UNI[2505] := 16#6177;
   // UNI[2506] := 16#618B;
   // UNI[2507] := 16#618E;
   // UNI[2508] := 16#6194;
   // UNI[2509] := 16#619D;
   // UNI[2510] := 16#61A7;
   // UNI[2511] := 16#61A8;
   // UNI[2512] := 16#61A9;
   // UNI[2513] := 16#61AC;
   // UNI[2514] := 16#61B7;
   // UNI[2515] := 16#61BE;
   // UNI[2516] := 16#61C2;
   // UNI[2517] := 16#61C8;
   // UNI[2518] := 16#61CA;
   // UNI[2519] := 16#61CB;
   // UNI[2520] := 16#61D1;
   // UNI[2521] := 16#61D2;
   // UNI[2522] := 16#61D4;
   // UNI[2523] := 16#61E6;
   // UNI[2524] := 16#61F5;
   // UNI[2525] := 16#61FF;
   // UNI[2526] := 16#6206;
   // UNI[2527] := 16#6208;
   // UNI[2528] := 16#620A;
   // UNI[2529] := 16#620B;
   // UNI[2530] := 16#620C;
   // UNI[2531] := 16#620D;
   // UNI[2532] := 16#620E;
   // UNI[2533] := 16#620F;
   // UNI[2534] := 16#6210;
   // UNI[2535] := 16#6211;
   // UNI[2536] := 16#6212;
   // UNI[2537] := 16#6215;
   // UNI[2538] := 16#6216;
   // UNI[2539] := 16#6217;
   // UNI[2540] := 16#6218;
   // UNI[2541] := 16#621A;
   // UNI[2542] := 16#621B;
   // UNI[2543] := 16#621F;
   // UNI[2544] := 16#6221;
   // UNI[2545] := 16#6222;
   // UNI[2546] := 16#6224;
   // UNI[2547] := 16#6225;
   // UNI[2548] := 16#622A;
   // UNI[2549] := 16#622C;
   // UNI[2550] := 16#622E;
   // UNI[2551] := 16#6233;
   // UNI[2552] := 16#6234;
   // UNI[2553] := 16#6237;
   // UNI[2554] := 16#623D;
   // UNI[2555] := 16#623E;
   // UNI[2556] := 16#623F;
   // UNI[2557] := 16#6240;
   // UNI[2558] := 16#6241;
   // UNI[2559] := 16#6243;
   // UNI[2560] := 16#6247;
   // UNI[2561] := 16#6248;
   // UNI[2562] := 16#6249;
   // UNI[2563] := 16#624B;
   // UNI[2564] := 16#624C;
   // UNI[2565] := 16#624D;
   // UNI[2566] := 16#624E;
   // UNI[2567] := 16#6251;
   // UNI[2568] := 16#6252;
   // UNI[2569] := 16#6253;
   // UNI[2570] := 16#6254;
   // UNI[2571] := 16#6258;
   // UNI[2572] := 16#625B;
   // UNI[2573] := 16#6263;
   // UNI[2574] := 16#6266;
   // UNI[2575] := 16#6267;
   // UNI[2576] := 16#6269;
   // UNI[2577] := 16#626A;
   // UNI[2578] := 16#626B;
   // UNI[2579] := 16#626C;
   // UNI[2580] := 16#626D;
   // UNI[2581] := 16#626E;
   // UNI[2582] := 16#626F;
   // UNI[2583] := 16#6270;
   // UNI[2584] := 16#6273;
   // UNI[2585] := 16#6276;
   // UNI[2586] := 16#6279;
   // UNI[2587] := 16#627C;
   // UNI[2588] := 16#627E;
   // UNI[2589] := 16#627F;
   // UNI[2590] := 16#6280;
   // UNI[2591] := 16#6284;
   // UNI[2592] := 16#6289;
   // UNI[2593] := 16#628A;
   // UNI[2594] := 16#6291;
   // UNI[2595] := 16#6292;
   // UNI[2596] := 16#6293;
   // UNI[2597] := 16#6295;
   // UNI[2598] := 16#6296;
   // UNI[2599] := 16#6297;
   // UNI[2600] := 16#6298;
   // UNI[2601] := 16#629A;
   // UNI[2602] := 16#629B;
   // UNI[2603] := 16#629F;
   // UNI[2604] := 16#62A0;
   // UNI[2605] := 16#62A1;
   // UNI[2606] := 16#62A2;
   // UNI[2607] := 16#62A4;
   // UNI[2608] := 16#62A5;
   // UNI[2609] := 16#62A8;
   // UNI[2610] := 16#62AB;
   // UNI[2611] := 16#62AC;
   // UNI[2612] := 16#62B1;
   // UNI[2613] := 16#62B5;
   // UNI[2614] := 16#62B9;
   // UNI[2615] := 16#62BB;
   // UNI[2616] := 16#62BC;
   // UNI[2617] := 16#62BD;
   // UNI[2618] := 16#62BF;
   // UNI[2619] := 16#62C2;
   // UNI[2620] := 16#62C4;
   // UNI[2621] := 16#62C5;
   // UNI[2622] := 16#62C6;
   // UNI[2623] := 16#62C7;
   // UNI[2624] := 16#62C8;
   // UNI[2625] := 16#62C9;
   // UNI[2626] := 16#62CA;
   // UNI[2627] := 16#62CC;
   // UNI[2628] := 16#62CD;
   // UNI[2629] := 16#62CE;
   // UNI[2630] := 16#62D0;
   // UNI[2631] := 16#62D2;
   // UNI[2632] := 16#62D3;
   // UNI[2633] := 16#62D4;
   // UNI[2634] := 16#62D6;
   // UNI[2635] := 16#62D7;
   // UNI[2636] := 16#62D8;
   // UNI[2637] := 16#62D9;
   // UNI[2638] := 16#62DA;
   // UNI[2639] := 16#62DB;
   // UNI[2640] := 16#62DC;
   // UNI[2641] := 16#62DF;
   // UNI[2642] := 16#62E2;
   // UNI[2643] := 16#62E3;
   // UNI[2644] := 16#62E5;
   // UNI[2645] := 16#62E6;
   // UNI[2646] := 16#62E7;
   // UNI[2647] := 16#62E8;
   // UNI[2648] := 16#62E9;
   // UNI[2649] := 16#62EC;
   // UNI[2650] := 16#62ED;
   // UNI[2651] := 16#62EE;
   // UNI[2652] := 16#62EF;
   // UNI[2653] := 16#62F1;
   // UNI[2654] := 16#62F3;
   // UNI[2655] := 16#62F4;
   // UNI[2656] := 16#62F6;
   // UNI[2657] := 16#62F7;
   // UNI[2658] := 16#62FC;
   // UNI[2659] := 16#62FD;
   // UNI[2660] := 16#62FE;
   // UNI[2661] := 16#62FF;
   // UNI[2662] := 16#6301;
   // UNI[2663] := 16#6302;
   // UNI[2664] := 16#6307;
   // UNI[2665] := 16#6308;
   // UNI[2666] := 16#6309;
   // UNI[2667] := 16#630E;
   // UNI[2668] := 16#6311;
   // UNI[2669] := 16#6316;
   // UNI[2670] := 16#631A;
   // UNI[2671] := 16#631B;
   // UNI[2672] := 16#631D;
   // UNI[2673] := 16#631E;
   // UNI[2674] := 16#631F;
   // UNI[2675] := 16#6320;
   // UNI[2676] := 16#6321;
   // UNI[2677] := 16#6322;
   // UNI[2678] := 16#6323;
   // UNI[2679] := 16#6324;
   // UNI[2680] := 16#6325;
   // UNI[2681] := 16#6328;
   // UNI[2682] := 16#632A;
   // UNI[2683] := 16#632B;
   // UNI[2684] := 16#632F;
   // UNI[2685] := 16#6332;
   // UNI[2686] := 16#6339;
   // UNI[2687] := 16#633A;
   // UNI[2688] := 16#633D;
   // UNI[2689] := 16#6342;
   // UNI[2690] := 16#6343;
   // UNI[2691] := 16#6345;
   // UNI[2692] := 16#6346;
   // UNI[2693] := 16#6349;
   // UNI[2694] := 16#634B;
   // UNI[2695] := 16#634C;
   // UNI[2696] := 16#634D;
   // UNI[2697] := 16#634E;
   // UNI[2698] := 16#634F;
   // UNI[2699] := 16#6350;
   // UNI[2700] := 16#6355;
   // UNI[2701] := 16#635E;
   // UNI[2702] := 16#635F;
   // UNI[2703] := 16#6361;
   // UNI[2704] := 16#6362;
   // UNI[2705] := 16#6363;
   // UNI[2706] := 16#6367;
   // UNI[2707] := 16#6369;
   // UNI[2708] := 16#636D;
   // UNI[2709] := 16#636E;
   // UNI[2710] := 16#6371;
   // UNI[2711] := 16#6376;
   // UNI[2712] := 16#6377;
   // UNI[2713] := 16#637A;
   // UNI[2714] := 16#637B;
   // UNI[2715] := 16#6380;
   // UNI[2716] := 16#6382;
   // UNI[2717] := 16#6387;
   // UNI[2718] := 16#6388;
   // UNI[2719] := 16#6389;
   // UNI[2720] := 16#638A;
   // UNI[2721] := 16#638C;
   // UNI[2722] := 16#638E;
   // UNI[2723] := 16#638F;
   // UNI[2724] := 16#6390;
   // UNI[2725] := 16#6392;
   // UNI[2726] := 16#6396;
   // UNI[2727] := 16#6398;
   // UNI[2728] := 16#63A0;
   // UNI[2729] := 16#63A2;
   // UNI[2730] := 16#63A3;
   // UNI[2731] := 16#63A5;
   // UNI[2732] := 16#63A7;
   // UNI[2733] := 16#63A8;
   // UNI[2734] := 16#63A9;
   // UNI[2735] := 16#63AA;
   // UNI[2736] := 16#63AC;
   // UNI[2737] := 16#63AD;
   // UNI[2738] := 16#63AE;
   // UNI[2739] := 16#63B0;
   // UNI[2740] := 16#63B3;
   // UNI[2741] := 16#63B4;
   // UNI[2742] := 16#63B7;
   // UNI[2743] := 16#63B8;
   // UNI[2744] := 16#63BA;
   // UNI[2745] := 16#63BC;
   // UNI[2746] := 16#63BE;
   // UNI[2747] := 16#63C4;
   // UNI[2748] := 16#63C6;
   // UNI[2749] := 16#63C9;
   // UNI[2750] := 16#63CD;
   // UNI[2751] := 16#63CE;
   // UNI[2752] := 16#63CF;
   // UNI[2753] := 16#63D0;
   // UNI[2754] := 16#63D2;
   // UNI[2755] := 16#63D6;
   // UNI[2756] := 16#63DE;
   // UNI[2757] := 16#63E0;
   // UNI[2758] := 16#63E1;
   // UNI[2759] := 16#63E3;
   // UNI[2760] := 16#63E9;
   // UNI[2761] := 16#63EA;
   // UNI[2762] := 16#63ED;
   // UNI[2763] := 16#63F2;
   // UNI[2764] := 16#63F4;
   // UNI[2765] := 16#63F6;
   // UNI[2766] := 16#63F8;
   // UNI[2767] := 16#63FD;
   // UNI[2768] := 16#63FF;
   // UNI[2769] := 16#6400;
   // UNI[2770] := 16#6401;
   // UNI[2771] := 16#6402;
   // UNI[2772] := 16#6405;
   // UNI[2773] := 16#640B;
   // UNI[2774] := 16#640C;
   // UNI[2775] := 16#640F;
   // UNI[2776] := 16#6410;
   // UNI[2777] := 16#6413;
   // UNI[2778] := 16#6414;
   // UNI[2779] := 16#641B;
   // UNI[2780] := 16#641C;
   // UNI[2781] := 16#641E;
   // UNI[2782] := 16#6420;
   // UNI[2783] := 16#6421;
   // UNI[2784] := 16#6426;
   // UNI[2785] := 16#642A;
   // UNI[2786] := 16#642C;
   // UNI[2787] := 16#642D;
   // UNI[2788] := 16#6434;
   // UNI[2789] := 16#643A;
   // UNI[2790] := 16#643D;
   // UNI[2791] := 16#643F;
   // UNI[2792] := 16#6441;
   // UNI[2793] := 16#6444;
   // UNI[2794] := 16#6445;
   // UNI[2795] := 16#6446;
   // UNI[2796] := 16#6447;
   // UNI[2797] := 16#6448;
   // UNI[2798] := 16#644A;
   // UNI[2799] := 16#6452;
   // UNI[2800] := 16#6454;
   // UNI[2801] := 16#6458;
   // UNI[2802] := 16#645E;
   // UNI[2803] := 16#6467;
   // UNI[2804] := 16#6469;
   // UNI[2805] := 16#646D;
   // UNI[2806] := 16#6478;
   // UNI[2807] := 16#6479;
   // UNI[2808] := 16#647A;
   // UNI[2809] := 16#6482;
   // UNI[2810] := 16#6484;
   // UNI[2811] := 16#6485;
   // UNI[2812] := 16#6487;
   // UNI[2813] := 16#6491;
   // UNI[2814] := 16#6492;
   // UNI[2815] := 16#6495;
   // UNI[2816] := 16#6496;
   // UNI[2817] := 16#6499;
   // UNI[2818] := 16#649E;
   // UNI[2819] := 16#64A4;
   // UNI[2820] := 16#64A9;
   // UNI[2821] := 16#64AC;
   // UNI[2822] := 16#64AD;
   // UNI[2823] := 16#64AE;
   // UNI[2824] := 16#64B0;
   // UNI[2825] := 16#64B5;
   // UNI[2826] := 16#64B7;
   // UNI[2827] := 16#64B8;
   // UNI[2828] := 16#64BA;
   // UNI[2829] := 16#64BC;
   // UNI[2830] := 16#64C0;
   // UNI[2831] := 16#64C2;
   // UNI[2832] := 16#64C5;
   // UNI[2833] := 16#64CD;
   // UNI[2834] := 16#64CE;
   // UNI[2835] := 16#64D0;
   // UNI[2836] := 16#64D2;
   // UNI[2837] := 16#64D7;
   // UNI[2838] := 16#64D8;
   // UNI[2839] := 16#64DE;
   // UNI[2840] := 16#64E2;
   // UNI[2841] := 16#64E4;
   // UNI[2842] := 16#64E6;
   // UNI[2843] := 16#6500;
   // UNI[2844] := 16#6509;
   // UNI[2845] := 16#6512;
   // UNI[2846] := 16#6518;
   // UNI[2847] := 16#6525;
   // UNI[2848] := 16#652B;
   // UNI[2849] := 16#652E;
   // UNI[2850] := 16#652F;
   // UNI[2851] := 16#6534;
   // UNI[2852] := 16#6535;
   // UNI[2853] := 16#6536;
   // UNI[2854] := 16#6538;
   // UNI[2855] := 16#6539;
   // UNI[2856] := 16#653B;
   // UNI[2857] := 16#653E;
   // UNI[2858] := 16#653F;
   // UNI[2859] := 16#6545;
   // UNI[2860] := 16#6548;
   // UNI[2861] := 16#6549;
   // UNI[2862] := 16#654C;
   // UNI[2863] := 16#654F;
   // UNI[2864] := 16#6551;
   // UNI[2865] := 16#6555;
   // UNI[2866] := 16#6556;
   // UNI[2867] := 16#6559;
   // UNI[2868] := 16#655B;
   // UNI[2869] := 16#655D;
   // UNI[2870] := 16#655E;
   // UNI[2871] := 16#6562;
   // UNI[2872] := 16#6563;
   // UNI[2873] := 16#6566;
   // UNI[2874] := 16#656B;
   // UNI[2875] := 16#656C;
   // UNI[2876] := 16#6570;
   // UNI[2877] := 16#6572;
   // UNI[2878] := 16#6574;
   // UNI[2879] := 16#6577;
   // UNI[2880] := 16#6587;
   // UNI[2881] := 16#658B;
   // UNI[2882] := 16#658C;
   // UNI[2883] := 16#6590;
   // UNI[2884] := 16#6591;
   // UNI[2885] := 16#6593;
   // UNI[2886] := 16#6597;
   // UNI[2887] := 16#6599;
   // UNI[2888] := 16#659B;
   // UNI[2889] := 16#659C;
   // UNI[2890] := 16#659F;
   // UNI[2891] := 16#65A1;
   // UNI[2892] := 16#65A4;
   // UNI[2893] := 16#65A5;
   // UNI[2894] := 16#65A7;
   // UNI[2895] := 16#65A9;
   // UNI[2896] := 16#65AB;
   // UNI[2897] := 16#65AD;
   // UNI[2898] := 16#65AF;
   // UNI[2899] := 16#65B0;
   // UNI[2900] := 16#65B9;
   // UNI[2901] := 16#65BC;
   // UNI[2902] := 16#65BD;
   // UNI[2903] := 16#65C1;
   // UNI[2904] := 16#65C3;
   // UNI[2905] := 16#65C4;
   // UNI[2906] := 16#65C5;
   // UNI[2907] := 16#65C6;
   // UNI[2908] := 16#65CB;
   // UNI[2909] := 16#65CC;
   // UNI[2910] := 16#65CE;
   // UNI[2911] := 16#65CF;
   // UNI[2912] := 16#65D2;
   // UNI[2913] := 16#65D6;
   // UNI[2914] := 16#65D7;
   // UNI[2915] := 16#65E0;
   // UNI[2916] := 16#65E2;
   // UNI[2917] := 16#65E5;
   // UNI[2918] := 16#65E6;
   // UNI[2919] := 16#65E7;
   // UNI[2920] := 16#65E8;
   // UNI[2921] := 16#65E9;
   // UNI[2922] := 16#65EC;
   // UNI[2923] := 16#65ED;
   // UNI[2924] := 16#65EE;
   // UNI[2925] := 16#65EF;
   // UNI[2926] := 16#65F0;
   // UNI[2927] := 16#65F1;
   // UNI[2928] := 16#65F6;
   // UNI[2929] := 16#65F7;
   // UNI[2930] := 16#65FA;
   // UNI[2931] := 16#6600;
   // UNI[2932] := 16#6602;
   // UNI[2933] := 16#6603;
   // UNI[2934] := 16#6606;
   // UNI[2935] := 16#660A;
   // UNI[2936] := 16#660C;
   // UNI[2937] := 16#660E;
   // UNI[2938] := 16#660F;
   // UNI[2939] := 16#6613;
   // UNI[2940] := 16#6614;
   // UNI[2941] := 16#6615;
   // UNI[2942] := 16#6619;
   // UNI[2943] := 16#661D;
   // UNI[2944] := 16#661F;
   // UNI[2945] := 16#6620;
   // UNI[2946] := 16#6625;
   // UNI[2947] := 16#6627;
   // UNI[2948] := 16#6628;
   // UNI[2949] := 16#662D;
   // UNI[2950] := 16#662F;
   // UNI[2951] := 16#6631;
   // UNI[2952] := 16#6634;
   // UNI[2953] := 16#6635;
   // UNI[2954] := 16#6636;
   // UNI[2955] := 16#663C;
   // UNI[2956] := 16#663E;
   // UNI[2957] := 16#6641;
   // UNI[2958] := 16#6643;
   // UNI[2959] := 16#664B;
   // UNI[2960] := 16#664C;
   // UNI[2961] := 16#664F;
   // UNI[2962] := 16#6652;
   // UNI[2963] := 16#6653;
   // UNI[2964] := 16#6654;
   // UNI[2965] := 16#6655;
   // UNI[2966] := 16#6656;
   // UNI[2967] := 16#6657;
   // UNI[2968] := 16#665A;
   // UNI[2969] := 16#665F;
   // UNI[2970] := 16#6661;
   // UNI[2971] := 16#6664;
   // UNI[2972] := 16#6666;
   // UNI[2973] := 16#6668;
   // UNI[2974] := 16#666E;
   // UNI[2975] := 16#666F;
   // UNI[2976] := 16#6670;
   // UNI[2977] := 16#6674;
   // UNI[2978] := 16#6676;
   // UNI[2979] := 16#6677;
   // UNI[2980] := 16#667A;
   // UNI[2981] := 16#667E;
   // UNI[2982] := 16#6682;
   // UNI[2983] := 16#6684;
   // UNI[2984] := 16#6687;
   // UNI[2985] := 16#668C;
   // UNI[2986] := 16#6691;
   // UNI[2987] := 16#6696;
   // UNI[2988] := 16#6697;
   // UNI[2989] := 16#669D;
   // UNI[2990] := 16#66A7;
   // UNI[2991] := 16#66A8;
   // UNI[2992] := 16#66AE;
   // UNI[2993] := 16#66B4;
   // UNI[2994] := 16#66B9;
   // UNI[2995] := 16#66BE;
   // UNI[2996] := 16#66D9;
   // UNI[2997] := 16#66DB;
   // UNI[2998] := 16#66DC;
   // UNI[2999] := 16#66DD;
   // UNI[3000] := 16#66E6;
   // UNI[3001] := 16#66E9;
   // UNI[3002] := 16#66F0;
   // UNI[3003] := 16#66F2;
   // UNI[3004] := 16#66F3;
   // UNI[3005] := 16#66F4;
   // UNI[3006] := 16#66F7;
   // UNI[3007] := 16#66F9;
   // UNI[3008] := 16#66FC;
   // UNI[3009] := 16#66FE;
   // UNI[3010] := 16#66FF;
   // UNI[3011] := 16#6700;
   // UNI[3012] := 16#6708;
   // UNI[3013] := 16#6709;
   // UNI[3014] := 16#670A;
   // UNI[3015] := 16#670B;
   // UNI[3016] := 16#670D;
   // UNI[3017] := 16#6710;
   // UNI[3018] := 16#6714;
   // UNI[3019] := 16#6715;
   // UNI[3020] := 16#6717;
   // UNI[3021] := 16#671B;
   // UNI[3022] := 16#671D;
   // UNI[3023] := 16#671F;
   // UNI[3024] := 16#6726;
   // UNI[3025] := 16#6728;
   // UNI[3026] := 16#672A;
   // UNI[3027] := 16#672B;
   // UNI[3028] := 16#672C;
   // UNI[3029] := 16#672D;
   // UNI[3030] := 16#672F;
   // UNI[3031] := 16#6731;
   // UNI[3032] := 16#6734;
   // UNI[3033] := 16#6735;
   // UNI[3034] := 16#673A;
   // UNI[3035] := 16#673D;
   // UNI[3036] := 16#6740;
   // UNI[3037] := 16#6742;
   // UNI[3038] := 16#6743;
   // UNI[3039] := 16#6746;
   // UNI[3040] := 16#6748;
   // UNI[3041] := 16#6749;
   // UNI[3042] := 16#674C;
   // UNI[3043] := 16#674E;
   // UNI[3044] := 16#674F;
   // UNI[3045] := 16#6750;
   // UNI[3046] := 16#6751;
   // UNI[3047] := 16#6753;
   // UNI[3048] := 16#6756;
   // UNI[3049] := 16#675C;
   // UNI[3050] := 16#675E;
   // UNI[3051] := 16#675F;
   // UNI[3052] := 16#6760;
   // UNI[3053] := 16#6761;
   // UNI[3054] := 16#6765;
   // UNI[3055] := 16#6768;
   // UNI[3056] := 16#6769;
   // UNI[3057] := 16#676A;
   // UNI[3058] := 16#676D;
   // UNI[3059] := 16#676F;
   // UNI[3060] := 16#6770;
   // UNI[3061] := 16#6772;
   // UNI[3062] := 16#6773;
   // UNI[3063] := 16#6775;
   // UNI[3064] := 16#6777;
   // UNI[3065] := 16#677C;
   // UNI[3066] := 16#677E;
   // UNI[3067] := 16#677F;
   // UNI[3068] := 16#6781;
   // UNI[3069] := 16#6784;
   // UNI[3070] := 16#6787;
   // UNI[3071] := 16#6789;
   // UNI[3072] := 16#678B;
   // UNI[3073] := 16#6790;
   // UNI[3074] := 16#6795;
   // UNI[3075] := 16#6797;
   // UNI[3076] := 16#6798;
   // UNI[3077] := 16#679A;
   // UNI[3078] := 16#679C;
   // UNI[3079] := 16#679D;
   // UNI[3080] := 16#679E;
   // UNI[3081] := 16#67A2;
   // UNI[3082] := 16#67A3;
   // UNI[3083] := 16#67A5;
   // UNI[3084] := 16#67A7;
   // UNI[3085] := 16#67A8;
   // UNI[3086] := 16#67AA;
   // UNI[3087] := 16#67AB;
   // UNI[3088] := 16#67AD;
   // UNI[3089] := 16#67AF;
   // UNI[3090] := 16#67B0;
   // UNI[3091] := 16#67B3;
   // UNI[3092] := 16#67B5;
   // UNI[3093] := 16#67B6;
   // UNI[3094] := 16#67B7;
   // UNI[3095] := 16#67B8;
   // UNI[3096] := 16#67C1;
   // UNI[3097] := 16#67C3;
   // UNI[3098] := 16#67C4;
   // UNI[3099] := 16#67CF;
   // UNI[3100] := 16#67D0;
   // UNI[3101] := 16#67D1;
   // UNI[3102] := 16#67D2;
   // UNI[3103] := 16#67D3;
   // UNI[3104] := 16#67D4;
   // UNI[3105] := 16#67D8;
   // UNI[3106] := 16#67D9;
   // UNI[3107] := 16#67DA;
   // UNI[3108] := 16#67DC;
   // UNI[3109] := 16#67DD;
   // UNI[3110] := 16#67DE;
   // UNI[3111] := 16#67E0;
   // UNI[3112] := 16#67E2;
   // UNI[3113] := 16#67E5;
   // UNI[3114] := 16#67E9;
   // UNI[3115] := 16#67EC;
   // UNI[3116] := 16#67EF;
   // UNI[3117] := 16#67F0;
   // UNI[3118] := 16#67F1;
   // UNI[3119] := 16#67F3;
   // UNI[3120] := 16#67F4;
   // UNI[3121] := 16#67FD;
   // UNI[3122] := 16#67FF;
   // UNI[3123] := 16#6800;
   // UNI[3124] := 16#6805;
   // UNI[3125] := 16#6807;
   // UNI[3126] := 16#6808;
   // UNI[3127] := 16#6809;
   // UNI[3128] := 16#680A;
   // UNI[3129] := 16#680B;
   // UNI[3130] := 16#680C;
   // UNI[3131] := 16#680E;
   // UNI[3132] := 16#680F;
   // UNI[3133] := 16#6811;
   // UNI[3134] := 16#6813;
   // UNI[3135] := 16#6816;
   // UNI[3136] := 16#6817;
   // UNI[3137] := 16#681D;
   // UNI[3138] := 16#6821;
   // UNI[3139] := 16#6829;
   // UNI[3140] := 16#682A;
   // UNI[3141] := 16#6832;
   // UNI[3142] := 16#6833;
   // UNI[3143] := 16#6837;
   // UNI[3144] := 16#6838;
   // UNI[3145] := 16#6839;
   // UNI[3146] := 16#683C;
   // UNI[3147] := 16#683D;
   // UNI[3148] := 16#683E;
   // UNI[3149] := 16#6840;
   // UNI[3150] := 16#6841;
   // UNI[3151] := 16#6842;
   // UNI[3152] := 16#6843;
   // UNI[3153] := 16#6844;
   // UNI[3154] := 16#6845;
   // UNI[3155] := 16#6846;
   // UNI[3156] := 16#6848;
   // UNI[3157] := 16#6849;
   // UNI[3158] := 16#684A;
   // UNI[3159] := 16#684C;
   // UNI[3160] := 16#684E;
   // UNI[3161] := 16#6850;
   // UNI[3162] := 16#6851;
   // UNI[3163] := 16#6853;
   // UNI[3164] := 16#6854;
   // UNI[3165] := 16#6855;
   // UNI[3166] := 16#6860;
   // UNI[3167] := 16#6861;
   // UNI[3168] := 16#6862;
   // UNI[3169] := 16#6863;
   // UNI[3170] := 16#6864;
   // UNI[3171] := 16#6865;
   // UNI[3172] := 16#6866;
   // UNI[3173] := 16#6867;
   // UNI[3174] := 16#6868;
   // UNI[3175] := 16#6869;
   // UNI[3176] := 16#686B;
   // UNI[3177] := 16#6874;
   // UNI[3178] := 16#6876;
   // UNI[3179] := 16#6877;
   // UNI[3180] := 16#6881;
   // UNI[3181] := 16#6883;
   // UNI[3182] := 16#6885;
   // UNI[3183] := 16#6886;
   // UNI[3184] := 16#688F;
   // UNI[3185] := 16#6893;
   // UNI[3186] := 16#6897;
   // UNI[3187] := 16#68A2;
   // UNI[3188] := 16#68A6;
   // UNI[3189] := 16#68A7;
   // UNI[3190] := 16#68A8;
   // UNI[3191] := 16#68AD;
   // UNI[3192] := 16#68AF;
   // UNI[3193] := 16#68B0;
   // UNI[3194] := 16#68B3;
   // UNI[3195] := 16#68B5;
   // UNI[3196] := 16#68C0;
   // UNI[3197] := 16#68C2;
   // UNI[3198] := 16#68C9;
   // UNI[3199] := 16#68CB;
   // UNI[3200] := 16#68CD;
   // UNI[3201] := 16#68D2;
   // UNI[3202] := 16#68D5;
   // UNI[3203] := 16#68D8;
   // UNI[3204] := 16#68DA;
   // UNI[3205] := 16#68E0;
   // UNI[3206] := 16#68E3;
   // UNI[3207] := 16#68EE;
   // UNI[3208] := 16#68F0;
   // UNI[3209] := 16#68F1;
   // UNI[3210] := 16#68F5;
   // UNI[3211] := 16#68F9;
   // UNI[3212] := 16#68FA;
   // UNI[3213] := 16#68FC;
   // UNI[3214] := 16#6901;
   // UNI[3215] := 16#6905;
   // UNI[3216] := 16#690B;
   // UNI[3217] := 16#690D;
   // UNI[3218] := 16#690E;
   // UNI[3219] := 16#6910;
   // UNI[3220] := 16#6912;
   // UNI[3221] := 16#691F;
   // UNI[3222] := 16#6920;
   // UNI[3223] := 16#6924;
   // UNI[3224] := 16#692D;
   // UNI[3225] := 16#6930;
   // UNI[3226] := 16#6934;
   // UNI[3227] := 16#6939;
   // UNI[3228] := 16#693D;
   // UNI[3229] := 16#693F;
   // UNI[3230] := 16#6942;
   // UNI[3231] := 16#6954;
   // UNI[3232] := 16#6957;
   // UNI[3233] := 16#695A;
   // UNI[3234] := 16#695D;
   // UNI[3235] := 16#695E;
   // UNI[3236] := 16#6960;
   // UNI[3237] := 16#6963;
   // UNI[3238] := 16#6966;
   // UNI[3239] := 16#696B;
   // UNI[3240] := 16#696E;
   // UNI[3241] := 16#6971;
   // UNI[3242] := 16#6977;
   // UNI[3243] := 16#6978;
   // UNI[3244] := 16#6979;
   // UNI[3245] := 16#697C;
   // UNI[3246] := 16#6980;
   // UNI[3247] := 16#6982;
   // UNI[3248] := 16#6984;
   // UNI[3249] := 16#6986;
   // UNI[3250] := 16#6987;
   // UNI[3251] := 16#6988;
   // UNI[3252] := 16#6989;
   // UNI[3253] := 16#698D;
   // UNI[3254] := 16#6994;
   // UNI[3255] := 16#6995;
   // UNI[3256] := 16#6998;
   // UNI[3257] := 16#699B;
   // UNI[3258] := 16#699C;
   // UNI[3259] := 16#69A7;
   // UNI[3260] := 16#69A8;
   // UNI[3261] := 16#69AB;
   // UNI[3262] := 16#69AD;
   // UNI[3263] := 16#69B1;
   // UNI[3264] := 16#69B4;
   // UNI[3265] := 16#69B7;
   // UNI[3266] := 16#69BB;
   // UNI[3267] := 16#69C1;
   // UNI[3268] := 16#69CA;
   // UNI[3269] := 16#69CC;
   // UNI[3270] := 16#69CE;
   // UNI[3271] := 16#69D0;
   // UNI[3272] := 16#69D4;
   // UNI[3273] := 16#69DB;
   // UNI[3274] := 16#69DF;
   // UNI[3275] := 16#69E0;
   // UNI[3276] := 16#69ED;
   // UNI[3277] := 16#69F2;
   // UNI[3278] := 16#69FD;
   // UNI[3279] := 16#69FF;
   // UNI[3280] := 16#6A0A;
   // UNI[3281] := 16#6A17;
   // UNI[3282] := 16#6A18;
   // UNI[3283] := 16#6A1F;
   // UNI[3284] := 16#6A21;
   // UNI[3285] := 16#6A28;
   // UNI[3286] := 16#6A2A;
   // UNI[3287] := 16#6A2F;
   // UNI[3288] := 16#6A31;
   // UNI[3289] := 16#6A35;
   // UNI[3290] := 16#6A3D;
   // UNI[3291] := 16#6A3E;
   // UNI[3292] := 16#6A44;
   // UNI[3293] := 16#6A47;
   // UNI[3294] := 16#6A50;
   // UNI[3295] := 16#6A58;
   // UNI[3296] := 16#6A59;
   // UNI[3297] := 16#6A5B;
   // UNI[3298] := 16#6A61;
   // UNI[3299] := 16#6A65;
   // UNI[3300] := 16#6A71;
   // UNI[3301] := 16#6A79;
   // UNI[3302] := 16#6A7C;
   // UNI[3303] := 16#6A80;
   // UNI[3304] := 16#6A84;
   // UNI[3305] := 16#6A8E;
   // UNI[3306] := 16#6A90;
   // UNI[3307] := 16#6A91;
   // UNI[3308] := 16#6A97;
   // UNI[3309] := 16#6AA0;
   // UNI[3310] := 16#6AA9;
   // UNI[3311] := 16#6AAB;
   // UNI[3312] := 16#6AAC;
   // UNI[3313] := 16#6B20;
   // UNI[3314] := 16#6B21;
   // UNI[3315] := 16#6B22;
   // UNI[3316] := 16#6B23;
   // UNI[3317] := 16#6B24;
   // UNI[3318] := 16#6B27;
   // UNI[3319] := 16#6B32;
   // UNI[3320] := 16#6B37;
   // UNI[3321] := 16#6B39;
   // UNI[3322] := 16#6B3A;
   // UNI[3323] := 16#6B3E;
   // UNI[3324] := 16#6B43;
   // UNI[3325] := 16#6B46;
   // UNI[3326] := 16#6B47;
   // UNI[3327] := 16#6B49;
   // UNI[3328] := 16#6B4C;
   // UNI[3329] := 16#6B59;
   // UNI[3330] := 16#6B62;
   // UNI[3331] := 16#6B63;
   // UNI[3332] := 16#6B64;
   // UNI[3333] := 16#6B65;
   // UNI[3334] := 16#6B66;
   // UNI[3335] := 16#6B67;
   // UNI[3336] := 16#6B6A;
   // UNI[3337] := 16#6B79;
   // UNI[3338] := 16#6B7B;
   // UNI[3339] := 16#6B7C;
   // UNI[3340] := 16#6B81;
   // UNI[3341] := 16#6B82;
   // UNI[3342] := 16#6B83;
   // UNI[3343] := 16#6B84;
   // UNI[3344] := 16#6B86;
   // UNI[3345] := 16#6B87;
   // UNI[3346] := 16#6B89;
   // UNI[3347] := 16#6B8A;
   // UNI[3348] := 16#6B8B;
   // UNI[3349] := 16#6B8D;
   // UNI[3350] := 16#6B92;
   // UNI[3351] := 16#6B93;
   // UNI[3352] := 16#6B96;
   // UNI[3353] := 16#6B9A;
   // UNI[3354] := 16#6B9B;
   // UNI[3355] := 16#6BA1;
   // UNI[3356] := 16#6BAA;
   // UNI[3357] := 16#6BB3;
   // UNI[3358] := 16#6BB4;
   // UNI[3359] := 16#6BB5;
   // UNI[3360] := 16#6BB7;
   // UNI[3361] := 16#6BBF;
   // UNI[3362] := 16#6BC1;
   // UNI[3363] := 16#6BC2;
   // UNI[3364] := 16#6BC5;
   // UNI[3365] := 16#6BCB;
   // UNI[3366] := 16#6BCD;
   // UNI[3367] := 16#6BCF;
   // UNI[3368] := 16#6BD2;
   // UNI[3369] := 16#6BD3;
   // UNI[3370] := 16#6BD4;
   // UNI[3371] := 16#6BD5;
   // UNI[3372] := 16#6BD6;
   // UNI[3373] := 16#6BD7;
   // UNI[3374] := 16#6BD9;
   // UNI[3375] := 16#6BDB;
   // UNI[3376] := 16#6BE1;
   // UNI[3377] := 16#6BEA;
   // UNI[3378] := 16#6BEB;
   // UNI[3379] := 16#6BEF;
   // UNI[3380] := 16#6BF3;
   // UNI[3381] := 16#6BF5;
   // UNI[3382] := 16#6BF9;
   // UNI[3383] := 16#6BFD;
   // UNI[3384] := 16#6C05;
   // UNI[3385] := 16#6C06;
   // UNI[3386] := 16#6C07;
   // UNI[3387] := 16#6C0D;
   // UNI[3388] := 16#6C0F;
   // UNI[3389] := 16#6C10;
   // UNI[3390] := 16#6C11;
   // UNI[3391] := 16#6C13;
   // UNI[3392] := 16#6C14;
   // UNI[3393] := 16#6C15;
   // UNI[3394] := 16#6C16;
   // UNI[3395] := 16#6C18;
   // UNI[3396] := 16#6C19;
   // UNI[3397] := 16#6C1A;
   // UNI[3398] := 16#6C1B;
   // UNI[3399] := 16#6C1F;
   // UNI[3400] := 16#6C21;
   // UNI[3401] := 16#6C22;
   // UNI[3402] := 16#6C24;
   // UNI[3403] := 16#6C26;
   // UNI[3404] := 16#6C27;
   // UNI[3405] := 16#6C28;
   // UNI[3406] := 16#6C29;
   // UNI[3407] := 16#6C2A;
   // UNI[3408] := 16#6C2E;
   // UNI[3409] := 16#6C2F;
   // UNI[3410] := 16#6C30;
   // UNI[3411] := 16#6C32;
   // UNI[3412] := 16#6C34;
   // UNI[3413] := 16#6C35;
   // UNI[3414] := 16#6C38;
   // UNI[3415] := 16#6C3D;
   // UNI[3416] := 16#6C40;
   // UNI[3417] := 16#6C41;
   // UNI[3418] := 16#6C42;
   // UNI[3419] := 16#6C46;
   // UNI[3420] := 16#6C47;
   // UNI[3421] := 16#6C49;
   // UNI[3422] := 16#6C4A;
   // UNI[3423] := 16#6C50;
   // UNI[3424] := 16#6C54;
   // UNI[3425] := 16#6C55;
   // UNI[3426] := 16#6C57;
   // UNI[3427] := 16#6C5B;
   // UNI[3428] := 16#6C5C;
   // UNI[3429] := 16#6C5D;
   // UNI[3430] := 16#6C5E;
   // UNI[3431] := 16#6C5F;
   // UNI[3432] := 16#6C60;
   // UNI[3433] := 16#6C61;
   // UNI[3434] := 16#6C64;
   // UNI[3435] := 16#6C68;
   // UNI[3436] := 16#6C69;
   // UNI[3437] := 16#6C6A;
   // UNI[3438] := 16#6C70;
   // UNI[3439] := 16#6C72;
   // UNI[3440] := 16#6C74;
   // UNI[3441] := 16#6C76;
   // UNI[3442] := 16#6C79;
   // UNI[3443] := 16#6C7D;
   // UNI[3444] := 16#6C7E;
   // UNI[3445] := 16#6C81;
   // UNI[3446] := 16#6C82;
   // UNI[3447] := 16#6C83;
   // UNI[3448] := 16#6C85;
   // UNI[3449] := 16#6C86;
   // UNI[3450] := 16#6C88;
   // UNI[3451] := 16#6C89;
   // UNI[3452] := 16#6C8C;
   // UNI[3453] := 16#6C8F;
   // UNI[3454] := 16#6C90;
   // UNI[3455] := 16#6C93;
   // UNI[3456] := 16#6C94;
   // UNI[3457] := 16#6C99;
   // UNI[3458] := 16#6C9B;
   // UNI[3459] := 16#6C9F;
   // UNI[3460] := 16#6CA1;
   // UNI[3461] := 16#6CA3;
   // UNI[3462] := 16#6CA4;
   // UNI[3463] := 16#6CA5;
   // UNI[3464] := 16#6CA6;
   // UNI[3465] := 16#6CA7;
   // UNI[3466] := 16#6CA9;
   // UNI[3467] := 16#6CAA;
   // UNI[3468] := 16#6CAB;
   // UNI[3469] := 16#6CAD;
   // UNI[3470] := 16#6CAE;
   // UNI[3471] := 16#6CB1;
   // UNI[3472] := 16#6CB2;
   // UNI[3473] := 16#6CB3;
   // UNI[3474] := 16#6CB8;
   // UNI[3475] := 16#6CB9;
   // UNI[3476] := 16#6CBB;
   // UNI[3477] := 16#6CBC;
   // UNI[3478] := 16#6CBD;
   // UNI[3479] := 16#6CBE;
   // UNI[3480] := 16#6CBF;
   // UNI[3481] := 16#6CC4;
   // UNI[3482] := 16#6CC5;
   // UNI[3483] := 16#6CC9;
   // UNI[3484] := 16#6CCA;
   // UNI[3485] := 16#6CCC;
   // UNI[3486] := 16#6CD0;
   // UNI[3487] := 16#6CD3;
   // UNI[3488] := 16#6CD4;
   // UNI[3489] := 16#6CD5;
   // UNI[3490] := 16#6CD6;
   // UNI[3491] := 16#6CD7;
   // UNI[3492] := 16#6CDB;
   // UNI[3493] := 16#6CDE;
   // UNI[3494] := 16#6CE0;
   // UNI[3495] := 16#6CE1;
   // UNI[3496] := 16#6CE2;
   // UNI[3497] := 16#6CE3;
   // UNI[3498] := 16#6CE5;
   // UNI[3499] := 16#6CE8;
   // UNI[3500] := 16#6CEA;
   // UNI[3501] := 16#6CEB;
   // UNI[3502] := 16#6CEE;
   // UNI[3503] := 16#6CEF;
   // UNI[3504] := 16#6CF0;
   // UNI[3505] := 16#6CF1;
   // UNI[3506] := 16#6CF3;
   // UNI[3507] := 16#6CF5;
   // UNI[3508] := 16#6CF6;
   // UNI[3509] := 16#6CF7;
   // UNI[3510] := 16#6CF8;
   // UNI[3511] := 16#6CFA;
   // UNI[3512] := 16#6CFB;
   // UNI[3513] := 16#6CFC;
   // UNI[3514] := 16#6CFD;
   // UNI[3515] := 16#6CFE;
   // UNI[3516] := 16#6D01;
   // UNI[3517] := 16#6D04;
   // UNI[3518] := 16#6D07;
   // UNI[3519] := 16#6D0B;
   // UNI[3520] := 16#6D0C;
   // UNI[3521] := 16#6D0E;
   // UNI[3522] := 16#6D12;
   // UNI[3523] := 16#6D17;
   // UNI[3524] := 16#6D19;
   // UNI[3525] := 16#6D1A;
   // UNI[3526] := 16#6D1B;
   // UNI[3527] := 16#6D1E;
   // UNI[3528] := 16#6D25;
   // UNI[3529] := 16#6D27;
   // UNI[3530] := 16#6D2A;
   // UNI[3531] := 16#6D2B;
   // UNI[3532] := 16#6D2E;
   // UNI[3533] := 16#6D31;
   // UNI[3534] := 16#6D32;
   // UNI[3535] := 16#6D33;
   // UNI[3536] := 16#6D35;
   // UNI[3537] := 16#6D39;
   // UNI[3538] := 16#6D3B;
   // UNI[3539] := 16#6D3C;
   // UNI[3540] := 16#6D3D;
   // UNI[3541] := 16#6D3E;
   // UNI[3542] := 16#6D41;
   // UNI[3543] := 16#6D43;
   // UNI[3544] := 16#6D45;
   // UNI[3545] := 16#6D46;
   // UNI[3546] := 16#6D47;
   // UNI[3547] := 16#6D48;
   // UNI[3548] := 16#6D4A;
   // UNI[3549] := 16#6D4B;
   // UNI[3550] := 16#6D4D;
   // UNI[3551] := 16#6D4E;
   // UNI[3552] := 16#6D4F;
   // UNI[3553] := 16#6D51;
   // UNI[3554] := 16#6D52;
   // UNI[3555] := 16#6D53;
   // UNI[3556] := 16#6D54;
   // UNI[3557] := 16#6D59;
   // UNI[3558] := 16#6D5A;
   // UNI[3559] := 16#6D5C;
   // UNI[3560] := 16#6D5E;
   // UNI[3561] := 16#6D60;
   // UNI[3562] := 16#6D63;
   // UNI[3563] := 16#6D66;
   // UNI[3564] := 16#6D69;
   // UNI[3565] := 16#6D6A;
   // UNI[3566] := 16#6D6E;
   // UNI[3567] := 16#6D6F;
   // UNI[3568] := 16#6D74;
   // UNI[3569] := 16#6D77;
   // UNI[3570] := 16#6D78;
   // UNI[3571] := 16#6D7C;
   // UNI[3572] := 16#6D82;
   // UNI[3573] := 16#6D85;
   // UNI[3574] := 16#6D88;
   // UNI[3575] := 16#6D89;
   // UNI[3576] := 16#6D8C;
   // UNI[3577] := 16#6D8E;
   // UNI[3578] := 16#6D91;
   // UNI[3579] := 16#6D93;
   // UNI[3580] := 16#6D94;
   // UNI[3581] := 16#6D95;
   // UNI[3582] := 16#6D9B;
   // UNI[3583] := 16#6D9D;
   // UNI[3584] := 16#6D9E;
   // UNI[3585] := 16#6D9F;
   // UNI[3586] := 16#6DA0;
   // UNI[3587] := 16#6DA1;
   // UNI[3588] := 16#6DA3;
   // UNI[3589] := 16#6DA4;
   // UNI[3590] := 16#6DA6;
   // UNI[3591] := 16#6DA7;
   // UNI[3592] := 16#6DA8;
   // UNI[3593] := 16#6DA9;
   // UNI[3594] := 16#6DAA;
   // UNI[3595] := 16#6DAB;
